LIN {X -102.468,Y -19.656,Z -60.794,A -90.000,B 90.000,C 0.000} C_DIS
LIN {X -102.647,Y -19.661,Z -60.638,A -90.000,B 90.000,C 0.000} C_DIS
LIN {X -103.007,Y -19.669,Z -60.305,A -90.000,B 90.000,C 0.000} C_DIS
LIN {X -103.209,Y -19.683,Z -60.113,A -90.000,B 90.000,C 0.000} C_DIS
LIN {X -103.495,Y -19.707,Z -59.844,A -90.000,B 90.000,C 0.000} C_DIS
LIN {X -103.666,Y -19.713,Z -59.667,A -90.000,B 90.000,C 0.000} C_DIS
LIN {X -103.779,Y -19.716,Z -59.547,A -90.000,B 90.000,C 0.000} C_DIS
LIN {X -103.860,Y -19.719,Z -59.459,A -90.000,B 90.000,C 0.000} C_DIS
LIN {X -104.495,Y -19.775,Z -58.745,A -90.000,B 90.000,C 0.000} C_DIS
LIN {X -104.595,Y -19.779,Z -58.623,A -90.000,B 90.000,C 0.000} C_DIS
LIN {X -104.835,Y -19.785,Z -58.316,A -90.000,B 90.000,C 0.000} C_DIS
LIN {X -104.978,Y -19.797,Z -58.132,A -90.000,B 90.000,C 0.000} C_DIS
LIN {X -105.043,Y -19.805,Z -58.047,A -90.000,B 90.000,C 0.000} C_DIS
LIN {X -105.125,Y -19.819,Z -57.934,A -90.000,B 90.000,C 0.000} C_DIS
LIN {X -105.385,Y -19.857,Z -57.556,A -90.000,B 90.000,C 0.000} C_DIS
LIN {X -105.527,Y -19.870,Z -57.329,A -90.000,B 90.000,C 0.000} C_DIS
LIN {X -105.764,Y -19.897,Z -56.936,A -90.000,B 90.000,C 0.000} C_DIS
LIN {X -105.854,Y -19.911,Z -56.776,A -90.000,B 90.000,C 0.000} C_DIS
LIN {X -105.917,Y -19.926,Z -56.657,A -90.000,B 90.000,C 0.000} C_DIS
LIN {X -105.996,Y -19.941,Z -56.500,A -90.000,B 90.000,C 0.000} C_DIS
LIN {X -106.032,Y -19.946,Z -56.422,A -90.000,B 90.000,C 0.000} C_DIS
LIN {X -106.214,Y -19.970,Z -56.038,A -90.000,B 90.000,C 0.000} C_DIS
LIN {X -106.380,Y -19.996,Z -55.650,A -90.000,B 90.000,C 0.000} C_DIS
LIN {X -106.472,Y -20.020,Z -55.411,A -90.000,B 90.000,C 0.000} C_DIS
LIN {X -106.494,Y -20.024,Z -55.349,A -90.000,B 90.000,C 0.000} C_DIS
LIN {X -106.535,Y -20.035,Z -55.220,A -90.000,B 90.000,C 0.000} C_DIS
LIN {X -106.617,Y -20.062,Z -54.946,A -90.000,B 90.000,C 0.000} C_DIS
LIN {X -106.692,Y -20.075,Z -54.624,A -90.000,B 90.000,C 0.000} C_DIS
LIN {X -106.760,Y -20.092,Z -54.341,A -90.000,B 90.000,C 0.000} C_DIS
LIN {X -106.862,Y -20.115,Z -53.878,A -90.000,B 90.000,C 0.000} C_DIS
LIN {X -106.884,Y -20.121,Z -53.754,A -90.000,B 90.000,C 0.000} C_DIS
LIN {X -106.893,Y -20.125,Z -53.683,A -90.000,B 90.000,C 0.000} C_DIS
LIN {X -106.930,Y -20.149,Z -53.353,A -90.000,B 90.000,C 0.000} C_DIS
LIN {X -106.945,Y -20.158,Z -53.148,A -90.000,B 90.000,C 0.000} C_DIS
LIN {X -106.963,Y -20.175,Z -52.914,A -90.000,B 90.000,C 0.000} C_DIS
LIN {X -106.986,Y -20.187,Z -52.670,A -90.000,B 90.000,C 0.000} C_DIS
LIN {X -106.991,Y -20.199,Z -52.434,A -90.000,B 90.000,C 0.000} C_DIS
LIN {X -106.989,Y -20.206,Z -52.353,A -90.000,B 90.000,C 0.000} C_DIS
LIN {X -106.977,Y -20.220,Z -52.109,A -90.000,B 90.000,C 0.000} C_DIS
LIN {X -106.972,Y -20.227,Z -51.945,A -90.000,B 90.000,C 0.000} C_DIS
LIN {X -106.965,Y -20.243,Z -51.722,A -90.000,B 90.000,C 0.000} C_DIS
LIN {X -106.951,Y -20.255,Z -51.466,A -90.000,B 90.000,C 0.000} C_DIS
LIN {X -106.935,Y -20.264,Z -51.321,A -90.000,B 90.000,C 0.000} C_DIS
LIN {X -106.911,Y -20.273,Z -51.181,A -90.000,B 90.000,C 0.000} C_DIS
LIN {X -106.852,Y -20.297,Z -50.866,A -90.000,B 90.000,C 0.000} C_DIS
LIN {X -106.771,Y -20.330,Z -50.476,A -90.000,B 90.000,C 0.000} C_DIS
LIN {X -106.685,Y -20.335,Z -50.140,A -90.000,B 90.000,C 0.000} C_DIS
LIN {X -106.782,Y -20.243,Z -49.888,A -90.000,B 90.000,C 0.000} C_DIS
LIN {X -106.856,Y -20.158,Z -49.671,A -90.000,B 90.000,C 0.000} C_DIS
LIN {X -106.932,Y -20.067,Z -49.428,A -90.000,B 90.000,C 0.000} C_DIS
LIN {X -106.948,Y -20.044,Z -49.370,A -90.000,B 90.000,C 0.000} C_DIS
LIN {X -106.980,Y -19.994,Z -49.227,A -90.000,B 90.000,C 0.000} C_DIS
LIN {X -107.015,Y -19.922,Z -49.018,A -90.000,B 90.000,C 0.000} C_DIS
LIN {X -107.031,Y -19.869,Z -48.872,A -90.000,B 90.000,C 0.000} C_DIS
LIN {X -107.043,Y -19.802,Z -48.689,A -90.000,B 90.000,C 0.000} C_DIS
LIN {X -107.043,Y -19.769,Z -48.600,A -90.000,B 90.000,C 0.000} C_DIS
LIN {X -107.040,Y -19.702,Z -48.416,A -90.000,B 90.000,C 0.000} C_DIS
LIN {X -107.158,Y -19.716,Z -48.219,A -90.000,B 90.000,C 0.000} C_DIS
LIN {X -107.387,Y -19.753,Z -47.792,A -90.000,B 90.000,C 0.000} C_DIS
LIN {X -107.530,Y -19.779,Z -47.517,A -90.000,B 90.000,C 0.000} C_DIS
LIN {X -107.589,Y -19.788,Z -47.393,A -90.000,B 90.000,C 0.000} C_DIS
LIN {X -107.781,Y -19.805,Z -46.947,A -90.000,B 90.000,C 0.000} C_DIS
LIN {X -107.936,Y -19.835,Z -46.542,A -90.000,B 90.000,C 0.000} C_DIS
LIN {X -108.076,Y -19.861,Z -46.147,A -90.000,B 90.000,C 0.000} C_DIS
LIN {X -108.110,Y -19.866,Z -46.039,A -90.000,B 90.000,C 0.000} C_DIS
LIN {X -108.258,Y -19.905,Z -45.517,A -90.000,B 90.000,C 0.000} C_DIS
LIN {X -108.292,Y -19.918,Z -45.382,A -90.000,B 90.000,C 0.000} C_DIS
LIN {X -108.367,Y -19.945,Z -44.989,A -90.000,B 90.000,C 0.000} C_DIS
LIN {X -108.401,Y -19.963,Z -44.786,A -90.000,B 90.000,C 0.000} C_DIS
LIN {X -108.450,Y -19.994,Z -44.452,A -90.000,B 90.000,C 0.000} C_DIS
LIN {X -108.458,Y -20.003,Z -44.374,A -90.000,B 90.000,C 0.000} C_DIS
LIN {X -108.475,Y -20.034,Z -44.027,A -90.000,B 90.000,C 0.000} C_DIS
LIN {X -108.482,Y -20.061,Z -43.676,A -90.000,B 90.000,C 0.000} C_DIS
LIN {X -108.481,Y -20.063,Z -43.623,A -90.000,B 90.000,C 0.000} C_DIS
LIN {X -108.472,Y -20.076,Z -43.437,A -90.000,B 90.000,C 0.000} C_DIS
LIN {X -108.460,Y -20.088,Z -43.312,A -90.000,B 90.000,C 0.000} C_DIS
LIN {X -108.430,Y -20.106,Z -43.070,A -90.000,B 90.000,C 0.000} C_DIS
LIN {X -108.391,Y -20.124,Z -42.770,A -90.000,B 90.000,C 0.000} C_DIS
LIN {X -108.369,Y -20.134,Z -42.620,A -90.000,B 90.000,C 0.000} C_DIS
LIN {X -108.351,Y -20.143,Z -42.521,A -90.000,B 90.000,C 0.000} C_DIS
LIN {X -108.295,Y -20.154,Z -42.273,A -90.000,B 90.000,C 0.000} C_DIS
LIN {X -108.254,Y -20.164,Z -42.113,A -90.000,B 90.000,C 0.000} C_DIS
LIN {X -108.187,Y -20.183,Z -41.874,A -90.000,B 90.000,C 0.000} C_DIS
LIN {X -108.175,Y -20.184,Z -41.836,A -90.000,B 90.000,C 0.000} C_DIS
LIN {X -108.036,Y -20.196,Z -41.450,A -90.000,B 90.000,C 0.000} C_DIS
LIN {X -107.992,Y -20.202,Z -41.337,A -90.000,B 90.000,C 0.000} C_DIS
LIN {X -107.941,Y -20.210,Z -41.219,A -90.000,B 90.000,C 0.000} C_DIS
LIN {X -107.830,Y -20.216,Z -40.993,A -90.000,B 90.000,C 0.000} C_DIS
LIN {X -107.652,Y -20.229,Z -40.655,A -90.000,B 90.000,C 0.000} C_DIS
LIN {X -107.557,Y -20.231,Z -40.499,A -90.000,B 90.000,C 0.000} C_DIS
LIN {X -107.486,Y -20.236,Z -40.390,A -90.000,B 90.000,C 0.000} C_DIS
LIN {X -107.378,Y -20.243,Z -40.218,A -90.000,B 90.000,C 0.000} C_DIS
LIN {X -107.336,Y -20.247,Z -40.156,A -90.000,B 90.000,C 0.000} C_DIS
LIN {X -107.134,Y -20.247,Z -39.892,A -90.000,B 90.000,C 0.000} C_DIS
LIN {X -106.995,Y -20.248,Z -39.727,A -90.000,B 90.000,C 0.000} C_DIS
LIN {X -106.913,Y -20.255,Z -39.638,A -90.000,B 90.000,C 0.000} C_DIS
LIN {X -106.815,Y -20.255,Z -39.541,A -90.000,B 90.000,C 0.000} C_DIS
LIN {X -106.736,Y -20.252,Z -39.457,A -90.000,B 90.000,C 0.000} C_DIS
LIN {X -106.666,Y -20.252,Z -39.388,A -90.000,B 90.000,C 0.000} C_DIS
LIN {X -106.465,Y -20.238,Z -39.204,A -90.000,B 90.000,C 0.000} C_DIS
LIN {X -106.419,Y -20.237,Z -39.161,A -90.000,B 90.000,C 0.000} C_DIS
LIN {X -106.281,Y -20.233,Z -39.052,A -90.000,B 90.000,C 0.000} C_DIS
LIN {X -106.141,Y -20.233,Z -38.949,A -90.000,B 90.000,C 0.000} C_DIS
LIN {X -106.028,Y -20.228,Z -38.869,A -90.000,B 90.000,C 0.000} C_DIS
LIN {X -105.932,Y -20.222,Z -38.807,A -90.000,B 90.000,C 0.000} C_DIS
LIN {X -105.709,Y -20.209,Z -38.671,A -90.000,B 90.000,C 0.000} C_DIS
LIN {X -105.617,Y -20.200,Z -38.618,A -90.000,B 90.000,C 0.000} C_DIS
LIN {X -105.493,Y -20.190,Z -38.549,A -90.000,B 90.000,C 0.000} C_DIS
LIN {X -105.295,Y -20.180,Z -38.450,A -90.000,B 90.000,C 0.000} C_DIS
LIN {X -105.169,Y -20.170,Z -38.390,A -90.000,B 90.000,C 0.000} C_DIS
LIN {X -104.969,Y -20.158,Z -38.302,A -90.000,B 90.000,C 0.000} C_DIS
LIN {X -104.908,Y -20.152,Z -38.281,A -90.000,B 90.000,C 0.000} C_DIS
LIN {X -104.636,Y -20.132,Z -38.197,A -90.000,B 90.000,C 0.000} C_DIS
LIN {X -104.324,Y -20.111,Z -38.104,A -90.000,B 90.000,C 0.000} C_DIS
LIN {X -104.248,Y -20.104,Z -38.084,A -90.000,B 90.000,C 0.000} C_DIS
LIN {X -104.041,Y -20.090,Z -38.032,A -90.000,B 90.000,C 0.000} C_DIS
LIN {X -103.918,Y -20.081,Z -38.000,A -90.000,B 90.000,C 0.000} C_DIS
LIN {X -103.778,Y -20.066,Z -37.966,A -90.000,B 90.000,C 0.000} C_DIS
LIN {X -103.743,Y -20.075,Z -37.948,A -90.000,B 90.000,C 0.000} C_DIS
LIN {X -103.593,Y -20.116,Z -37.876,A -90.000,B 90.000,C 0.000} C_DIS
LIN {X -103.525,Y -20.135,Z -37.847,A -90.000,B 90.000,C 0.000} C_DIS
LIN {X -103.189,Y -20.234,Z -37.708,A -90.000,B 90.000,C 0.000} C_DIS
LIN {X -103.098,Y -20.260,Z -37.678,A -90.000,B 90.000,C 0.000} C_DIS
LIN {X -102.820,Y -20.336,Z -37.593,A -90.000,B 90.000,C 0.000} C_DIS
LIN {X -102.445,Y -20.444,Z -37.498,A -90.000,B 90.000,C 0.000} C_DIS
LIN {X -102.298,Y -20.487,Z -37.465,A -90.000,B 90.000,C 0.000} C_DIS
LIN {X -102.220,Y -20.485,Z -37.368,A -90.000,B 90.000,C 0.000} C_DIS
LIN {X -102.027,Y -20.483,Z -37.139,A -90.000,B 90.000,C 0.000} C_DIS
LIN {X -101.812,Y -20.465,Z -36.903,A -90.000,B 90.000,C 0.000} C_DIS
LIN {X -101.694,Y -20.455,Z -36.777,A -90.000,B 90.000,C 0.000} C_DIS
LIN {X -101.599,Y -20.451,Z -36.687,A -90.000,B 90.000,C 0.000} C_DIS
LIN {X -101.321,Y -20.445,Z -36.439,A -90.000,B 90.000,C 0.000} C_DIS
LIN {X -101.201,Y -20.438,Z -36.339,A -90.000,B 90.000,C 0.000} C_DIS
LIN {X -100.770,Y -20.415,Z -35.994,A -90.000,B 90.000,C 0.000} C_DIS
LIN {X -100.652,Y -20.410,Z -35.905,A -90.000,B 90.000,C 0.000} C_DIS
LIN {X -100.499,Y -20.406,Z -35.797,A -90.000,B 90.000,C 0.000} C_DIS
LIN {X -100.151,Y -20.388,Z -35.556,A -90.000,B 90.000,C 0.000} C_DIS
LIN {X -99.916,Y -20.381,Z -35.405,A -90.000,B 90.000,C 0.000} C_DIS
LIN {X -99.744,Y -20.377,Z -35.300,A -90.000,B 90.000,C 0.000} C_DIS
LIN {X -99.281,Y -20.363,Z -35.024,A -90.000,B 90.000,C 0.000} C_DIS
LIN {X -98.910,Y -20.352,Z -34.805,A -90.000,B 90.000,C 0.000} C_DIS
LIN {X -98.295,Y -20.344,Z -34.463,A -90.000,B 90.000,C 0.000} C_DIS
LIN {X -97.990,Y -20.342,Z -34.302,A -90.000,B 90.000,C 0.000} C_DIS
LIN {X -97.805,Y -20.337,Z -34.195,A -90.000,B 90.000,C 0.000} C_DIS
LIN {X -97.584,Y -20.328,Z -34.071,A -90.000,B 90.000,C 0.000} C_DIS
LIN {X -97.137,Y -20.320,Z -33.838,A -90.000,B 90.000,C 0.000} C_DIS
LIN {X -96.832,Y -20.314,Z -33.683,A -90.000,B 90.000,C 0.000} C_DIS
LIN {X -96.610,Y -20.308,Z -33.567,A -90.000,B 90.000,C 0.000} C_DIS
LIN {X -96.600,Y -20.286,Z -33.521,A -90.000,B 90.000,C 0.000} C_DIS
LIN {X -96.618,Y -20.295,Z -33.331,A -90.000,B 90.000,C 0.000} C_DIS
LIN {X -96.627,Y -20.305,Z -33.207,A -90.000,B 90.000,C 0.000} C_DIS
LIN {X -96.630,Y -20.322,Z -33.062,A -90.000,B 90.000,C 0.000} C_DIS
LIN {X -96.627,Y -20.328,Z -32.959,A -90.000,B 90.000,C 0.000} C_DIS
LIN {X -96.631,Y -20.329,Z -32.851,A -90.000,B 90.000,C 0.000} C_DIS
LIN {X -96.632,Y -20.333,Z -32.719,A -90.000,B 90.000,C 0.000} C_DIS
LIN {X -96.627,Y -20.331,Z -32.618,A -90.000,B 90.000,C 0.000} C_DIS
LIN {X -96.607,Y -20.330,Z -32.367,A -90.000,B 90.000,C 0.000} C_DIS
LIN {X -96.588,Y -20.322,Z -32.206,A -90.000,B 90.000,C 0.000} C_DIS
LIN {X -96.575,Y -20.319,Z -32.113,A -90.000,B 90.000,C 0.000} C_DIS
LIN {X -96.549,Y -20.317,Z -31.978,A -90.000,B 90.000,C 0.000} C_DIS
LIN {X -96.525,Y -20.324,Z -31.864,A -90.000,B 90.000,C 0.000} C_DIS
LIN {X -96.472,Y -20.326,Z -31.649,A -90.000,B 90.000,C 0.000} C_DIS
LIN {X -96.439,Y -20.328,Z -31.525,A -90.000,B 90.000,C 0.000} C_DIS
LIN {X -96.403,Y -20.326,Z -31.420,A -90.000,B 90.000,C 0.000} C_DIS
LIN {X -96.330,Y -20.307,Z -31.149,A -90.000,B 90.000,C 0.000} C_DIS
LIN {X -96.289,Y -20.298,Z -31.020,A -90.000,B 90.000,C 0.000} C_DIS
LIN {X -96.223,Y -20.292,Z -30.847,A -90.000,B 90.000,C 0.000} C_DIS
LIN {X -96.154,Y -20.291,Z -30.672,A -90.000,B 90.000,C 0.000} C_DIS
LIN {X -96.118,Y -20.285,Z -30.589,A -90.000,B 90.000,C 0.000} C_DIS
LIN {X -96.058,Y -20.279,Z -30.460,A -90.000,B 90.000,C 0.000} C_DIS
LIN {X -96.010,Y -20.277,Z -30.369,A -90.000,B 90.000,C 0.000} C_DIS
LIN {X -95.824,Y -20.245,Z -29.966,A -90.000,B 90.000,C 0.000} C_DIS
LIN {X -95.770,Y -20.241,Z -29.860,A -90.000,B 90.000,C 0.000} C_DIS
LIN {X -95.637,Y -20.227,Z -29.641,A -90.000,B 90.000,C 0.000} C_DIS
LIN {X -95.523,Y -20.215,Z -29.457,A -90.000,B 90.000,C 0.000} C_DIS
LIN {X -95.471,Y -20.215,Z -29.381,A -90.000,B 90.000,C 0.000} C_DIS
LIN {X -95.353,Y -20.211,Z -29.196,A -90.000,B 90.000,C 0.000} C_DIS
LIN {X -95.243,Y -20.197,Z -29.034,A -90.000,B 90.000,C 0.000} C_DIS
LIN {X -95.164,Y -20.190,Z -28.926,A -90.000,B 90.000,C 0.000} C_DIS
LIN {X -94.971,Y -20.177,Z -28.684,A -90.000,B 90.000,C 0.000} C_DIS
LIN {X -94.863,Y -20.172,Z -28.548,A -90.000,B 90.000,C 0.000} C_DIS
LIN {X -94.731,Y -20.163,Z -28.412,A -90.000,B 90.000,C 0.000} C_DIS
LIN {X -94.601,Y -20.160,Z -28.288,A -90.000,B 90.000,C 0.000} C_DIS
LIN {X -94.475,Y -20.153,Z -28.171,A -90.000,B 90.000,C 0.000} C_DIS
LIN {X -94.314,Y -20.151,Z -28.021,A -90.000,B 90.000,C 0.000} C_DIS
LIN {X -94.055,Y -20.125,Z -27.801,A -90.000,B 90.000,C 0.000} C_DIS
LIN {X -93.954,Y -20.114,Z -27.720,A -90.000,B 90.000,C 0.000} C_DIS
LIN {X -93.785,Y -20.104,Z -27.590,A -90.000,B 90.000,C 0.000} C_DIS
LIN {X -93.556,Y -20.075,Z -27.428,A -90.000,B 90.000,C 0.000} C_DIS
LIN {X -93.439,Y -20.063,Z -27.351,A -90.000,B 90.000,C 0.000} C_DIS
LIN {X -93.127,Y -20.040,Z -27.158,A -90.000,B 90.000,C 0.000} C_DIS
LIN {X -93.022,Y -20.034,Z -27.096,A -90.000,B 90.000,C 0.000} C_DIS
LIN {X -92.971,Y -20.029,Z -27.070,A -90.000,B 90.000,C 0.000} C_DIS
LIN {X -92.805,Y -20.021,Z -26.987,A -90.000,B 90.000,C 0.000} C_DIS
LIN {X -92.331,Y -19.981,Z -26.769,A -90.000,B 90.000,C 0.000} C_DIS
LIN {X -91.928,Y -19.956,Z -26.589,A -90.000,B 90.000,C 0.000} C_DIS
LIN {X -91.695,Y -19.940,Z -26.497,A -90.000,B 90.000,C 0.000} C_DIS
LIN {X -91.552,Y -19.927,Z -26.445,A -90.000,B 90.000,C 0.000} C_DIS
LIN {X -91.434,Y -19.921,Z -26.407,A -90.000,B 90.000,C 0.000} C_DIS
LIN {X -91.264,Y -19.922,Z -26.345,A -90.000,B 90.000,C 0.000} C_DIS
LIN {X -91.192,Y -19.919,Z -26.315,A -90.000,B 90.000,C 0.000} C_DIS
LIN {X -91.034,Y -19.911,Z -26.253,A -90.000,B 90.000,C 0.000} C_DIS
LIN {X -90.902,Y -19.902,Z -26.204,A -90.000,B 90.000,C 0.000} C_DIS
LIN {X -90.698,Y -19.867,Z -26.116,A -90.000,B 90.000,C 0.000} C_DIS
LIN {X -90.661,Y -19.863,Z -26.098,A -90.000,B 90.000,C 0.000} C_DIS
LIN {X -90.314,Y -19.805,Z -25.911,A -90.000,B 90.000,C 0.000} C_DIS
LIN {X -90.185,Y -19.779,Z -25.852,A -90.000,B 90.000,C 0.000} C_DIS
LIN {X -90.105,Y -19.764,Z -25.809,A -90.000,B 90.000,C 0.000} C_DIS
LIN {X -89.802,Y -19.720,Z -25.651,A -90.000,B 90.000,C 0.000} C_DIS
LIN {X -89.689,Y -19.701,Z -25.598,A -90.000,B 90.000,C 0.000} C_DIS
LIN {X -89.546,Y -19.681,Z -25.525,A -90.000,B 90.000,C 0.000} C_DIS
LIN {X -89.281,Y -19.641,Z -25.389,A -90.000,B 90.000,C 0.000} C_DIS
LIN {X -89.187,Y -19.632,Z -25.335,A -90.000,B 90.000,C 0.000} C_DIS
LIN {X -88.817,Y -19.594,Z -25.143,A -90.000,B 90.000,C 0.000} C_DIS
LIN {X -88.591,Y -19.569,Z -25.028,A -90.000,B 90.000,C 0.000} C_DIS
LIN {X -88.410,Y -19.554,Z -24.924,A -90.000,B 90.000,C 0.000} C_DIS
LIN {X -88.172,Y -19.533,Z -24.792,A -90.000,B 90.000,C 0.000} C_DIS
LIN {X -88.036,Y -19.523,Z -24.707,A -90.000,B 90.000,C 0.000} C_DIS
LIN {X -87.575,Y -19.491,Z -24.432,A -90.000,B 90.000,C 0.000} C_DIS
LIN {X -87.416,Y -19.486,Z -24.324,A -90.000,B 90.000,C 0.000} C_DIS
LIN {X -87.164,Y -19.473,Z -24.150,A -90.000,B 90.000,C 0.000} C_DIS
LIN {X -86.793,Y -19.466,Z -23.855,A -90.000,B 90.000,C 0.000} C_DIS
LIN {X -86.730,Y -19.468,Z -23.795,A -90.000,B 90.000,C 0.000} C_DIS
LIN {X -86.537,Y -19.469,Z -23.611,A -90.000,B 90.000,C 0.000} C_DIS
LIN {X -86.318,Y -19.481,Z -23.370,A -90.000,B 90.000,C 0.000} C_DIS
LIN {X -86.206,Y -19.483,Z -23.245,A -90.000,B 90.000,C 0.000} C_DIS
LIN {X -85.931,Y -19.501,Z -22.900,A -90.000,B 90.000,C 0.000} C_DIS
LIN {X -85.450,Y -19.527,Z -22.280,A -90.000,B 90.000,C 0.000} C_DIS
LIN {X -84.861,Y -19.552,Z -21.540,A -90.000,B 90.000,C 0.000} C_DIS
LIN {X -84.646,Y -19.565,Z -21.273,A -90.000,B 90.000,C 0.000} C_DIS
LIN {X -84.419,Y -19.582,Z -20.981,A -90.000,B 90.000,C 0.000} C_DIS
LIN {X -84.355,Y -19.586,Z -20.904,A -90.000,B 90.000,C 0.000} C_DIS
LIN {X -84.280,Y -19.596,Z -20.802,A -90.000,B 90.000,C 0.000} C_DIS
LIN {X -84.210,Y -19.604,Z -20.710,A -90.000,B 90.000,C 0.000} C_DIS
LIN {X -84.113,Y -19.625,Z -20.561,A -90.000,B 90.000,C 0.000} C_DIS
LIN {X -83.875,Y -19.667,Z -20.229,A -90.000,B 90.000,C 0.000} C_DIS
LIN {X -83.761,Y -19.686,Z -20.089,A -90.000,B 90.000,C 0.000} C_DIS
LIN {X -83.565,Y -19.718,Z -19.855,A -90.000,B 90.000,C 0.000} C_DIS
LIN {X -83.405,Y -19.736,Z -19.685,A -90.000,B 90.000,C 0.000} C_DIS
LIN {X -83.151,Y -19.771,Z -19.426,A -90.000,B 90.000,C 0.000} C_DIS
LIN {X -83.000,Y -19.792,Z -19.277,A -90.000,B 90.000,C 0.000} C_DIS
LIN {X -82.917,Y -19.798,Z -19.205,A -90.000,B 90.000,C 0.000} C_DIS
LIN {X -82.679,Y -19.814,Z -18.999,A -90.000,B 90.000,C 0.000} C_DIS
LIN {X -82.618,Y -19.818,Z -18.951,A -90.000,B 90.000,C 0.000} C_DIS
LIN {X -82.353,Y -19.825,Z -18.759,A -90.000,B 90.000,C 0.000} C_DIS
LIN {X -82.249,Y -19.827,Z -18.688,A -90.000,B 90.000,C 0.000} C_DIS
LIN {X -82.022,Y -19.835,Z -18.556,A -90.000,B 90.000,C 0.000} C_DIS
LIN {X -81.744,Y -19.845,Z -18.402,A -90.000,B 90.000,C 0.000} C_DIS
LIN {X -81.591,Y -19.856,Z -18.324,A -90.000,B 90.000,C 0.000} C_DIS
LIN {X -81.356,Y -19.872,Z -18.218,A -90.000,B 90.000,C 0.000} C_DIS
LIN {X -80.963,Y -19.878,Z -18.067,A -90.000,B 90.000,C 0.000} C_DIS
LIN {X -80.823,Y -19.875,Z -18.019,A -90.000,B 90.000,C 0.000} C_DIS
LIN {X -80.687,Y -19.875,Z -17.978,A -90.000,B 90.000,C 0.000} C_DIS
LIN {X -80.483,Y -19.882,Z -17.921,A -90.000,B 90.000,C 0.000} C_DIS
LIN {X -80.143,Y -19.891,Z -17.838,A -90.000,B 90.000,C 0.000} C_DIS
LIN {X -80.074,Y -19.891,Z -17.824,A -90.000,B 90.000,C 0.000} C_DIS
LIN {X -79.971,Y -19.891,Z -17.810,A -90.000,B 90.000,C 0.000} C_DIS
LIN {X -79.718,Y -19.897,Z -17.779,A -90.000,B 90.000,C 0.000} C_DIS
LIN {X -79.322,Y -19.900,Z -17.738,A -90.000,B 90.000,C 0.000} C_DIS
LIN {X -79.150,Y -19.903,Z -17.721,A -90.000,B 90.000,C 0.000} C_DIS
LIN {X -79.012,Y -19.900,Z -17.715,A -90.000,B 90.000,C 0.000} C_DIS
LIN {X -78.774,Y -19.905,Z -17.713,A -90.000,B 90.000,C 0.000} C_DIS
LIN {X -78.599,Y -19.909,Z -17.717,A -90.000,B 90.000,C 0.000} C_DIS
LIN {X -78.403,Y -19.912,Z -17.728,A -90.000,B 90.000,C 0.000} C_DIS
LIN {X -78.089,Y -19.927,Z -17.753,A -90.000,B 90.000,C 0.000} C_DIS
LIN {X -77.678,Y -19.933,Z -17.797,A -90.000,B 90.000,C 0.000} C_DIS
LIN {X -77.525,Y -19.934,Z -17.822,A -90.000,B 90.000,C 0.000} C_DIS
LIN {X -77.266,Y -19.938,Z -17.869,A -90.000,B 90.000,C 0.000} C_DIS
LIN {X -76.923,Y -19.951,Z -17.940,A -90.000,B 90.000,C 0.000} C_DIS
LIN {X -76.818,Y -19.954,Z -17.966,A -90.000,B 90.000,C 0.000} C_DIS
LIN {X -76.561,Y -19.967,Z -18.034,A -90.000,B 90.000,C 0.000} C_DIS
LIN {X -76.281,Y -19.971,Z -18.121,A -90.000,B 90.000,C 0.000} C_DIS
LIN {X -75.975,Y -19.976,Z -18.219,A -90.000,B 90.000,C 0.000} C_DIS
LIN {X -75.734,Y -19.987,Z -18.303,A -90.000,B 90.000,C 0.000} C_DIS
LIN {X -75.635,Y -19.994,Z -18.339,A -90.000,B 90.000,C 0.000} C_DIS
LIN {X -75.465,Y -20.005,Z -18.409,A -90.000,B 90.000,C 0.000} C_DIS
LIN {X -74.762,Y -20.027,Z -18.725,A -90.000,B 90.000,C 0.000} C_DIS
LIN {X -74.605,Y -20.034,Z -18.800,A -90.000,B 90.000,C 0.000} C_DIS
LIN {X -74.394,Y -20.048,Z -18.911,A -90.000,B 90.000,C 0.000} C_DIS
LIN {X -74.268,Y -20.054,Z -18.979,A -90.000,B 90.000,C 0.000} C_DIS
LIN {X -73.804,Y -20.064,Z -19.251,A -90.000,B 90.000,C 0.000} C_DIS
LIN {X -73.492,Y -20.076,Z -19.444,A -90.000,B 90.000,C 0.000} C_DIS
LIN {X -72.936,Y -20.103,Z -19.799,A -90.000,B 90.000,C 0.000} C_DIS
LIN {X -72.712,Y -20.106,Z -19.949,A -90.000,B 90.000,C 0.000} C_DIS
LIN {X -72.234,Y -20.123,Z -20.285,A -90.000,B 90.000,C 0.000} C_DIS
LIN {X -71.884,Y -20.137,Z -20.537,A -90.000,B 90.000,C 0.000} C_DIS
LIN {X -71.462,Y -20.145,Z -20.864,A -90.000,B 90.000,C 0.000} C_DIS
LIN {X -71.236,Y -20.154,Z -21.049,A -90.000,B 90.000,C 0.000} C_DIS
LIN {X -70.880,Y -20.173,Z -21.348,A -90.000,B 90.000,C 0.000} C_DIS
LIN {X -70.783,Y -20.175,Z -21.433,A -90.000,B 90.000,C 0.000} C_DIS
LIN {X -70.418,Y -20.180,Z -21.756,A -90.000,B 90.000,C 0.000} C_DIS
LIN {X -70.128,Y -20.183,Z -22.043,A -90.000,B 90.000,C 0.000} C_DIS
LIN {X -69.442,Y -20.206,Z -22.752,A -90.000,B 90.000,C 0.000} C_DIS
LIN {X -69.187,Y -20.202,Z -23.032,A -90.000,B 90.000,C 0.000} C_DIS
LIN {X -69.083,Y -20.202,Z -23.159,A -90.000,B 90.000,C 0.000} C_DIS
LIN {X -68.869,Y -20.210,Z -23.438,A -90.000,B 90.000,C 0.000} C_DIS
LIN {X -68.637,Y -20.225,Z -23.754,A -90.000,B 90.000,C 0.000} C_DIS
LIN {X -68.583,Y -20.230,Z -23.831,A -90.000,B 90.000,C 0.000} C_DIS
LIN {X -68.309,Y -20.252,Z -24.250,A -90.000,B 90.000,C 0.000} C_DIS
LIN {X -68.204,Y -20.256,Z -24.417,A -90.000,B 90.000,C 0.000} C_DIS
LIN {X -68.032,Y -20.246,Z -24.710,A -90.000,B 90.000,C 0.000} C_DIS
LIN {X -67.865,Y -20.243,Z -25.017,A -90.000,B 90.000,C 0.000} C_DIS
LIN {X -67.828,Y -20.241,Z -25.087,A -90.000,B 90.000,C 0.000} C_DIS
LIN {X -67.749,Y -20.242,Z -25.253,A -90.000,B 90.000,C 0.000} C_DIS
LIN {X -67.626,Y -20.257,Z -25.556,A -90.000,B 90.000,C 0.000} C_DIS
LIN {X -67.456,Y -20.266,Z -26.002,A -90.000,B 90.000,C 0.000} C_DIS
LIN {X -67.395,Y -20.268,Z -26.166,A -90.000,B 90.000,C 0.000} C_DIS
LIN {X -67.219,Y -20.281,Z -26.690,A -90.000,B 90.000,C 0.000} C_DIS
LIN {X -67.180,Y -20.281,Z -26.813,A -90.000,B 90.000,C 0.000} C_DIS
LIN {X -67.098,Y -20.285,Z -27.099,A -90.000,B 90.000,C 0.000} C_DIS
LIN {X -67.045,Y -20.286,Z -27.302,A -90.000,B 90.000,C 0.000} C_DIS
LIN {X -66.996,Y -20.291,Z -27.515,A -90.000,B 90.000,C 0.000} C_DIS
LIN {X -66.968,Y -20.291,Z -27.645,A -90.000,B 90.000,C 0.000} C_DIS
LIN {X -66.922,Y -20.295,Z -27.887,A -90.000,B 90.000,C 0.000} C_DIS
LIN {X -66.829,Y -20.314,Z -28.354,A -90.000,B 90.000,C 0.000} C_DIS
LIN {X -66.764,Y -20.323,Z -28.692,A -90.000,B 90.000,C 0.000} C_DIS
LIN {X -66.683,Y -20.332,Z -29.124,A -90.000,B 90.000,C 0.000} C_DIS
LIN {X -66.657,Y -20.338,Z -29.304,A -90.000,B 90.000,C 0.000} C_DIS
LIN {X -66.626,Y -20.341,Z -29.467,A -90.000,B 90.000,C 0.000} C_DIS
LIN {X -66.435,Y -20.418,Z -30.349,A -90.000,B 90.000,C 0.000} C_DIS
LIN {X -66.338,Y -20.418,Z -30.590,A -90.000,B 90.000,C 0.000} C_DIS
LIN {X -66.194,Y -20.462,Z -30.893,A -90.000,B 90.000,C 0.000} C_DIS
LIN {X -66.076,Y -20.458,Z -31.015,A -90.000,B 90.000,C 0.000} C_DIS
LIN {X -65.600,Y -20.441,Z -31.509,A -90.000,B 90.000,C 0.000} C_DIS
LIN {X -65.490,Y -20.453,Z -31.618,A -90.000,B 90.000,C 0.000} C_DIS
LIN {X -64.665,Y -20.443,Z -32.167,A -90.000,B 90.000,C 0.000} C_DIS
LIN {X -64.188,Y -20.434,Z -32.479,A -90.000,B 90.000,C 0.000} C_DIS
LIN {X -63.993,Y -20.442,Z -32.599,A -90.000,B 90.000,C 0.000} C_DIS
LIN {X -62.272,Y -20.445,Z -33.500,A -90.000,B 90.000,C 0.000} C_DIS
LIN {X -61.786,Y -20.460,Z -33.747,A -90.000,B 90.000,C 0.000} C_DIS
LIN {X -61.215,Y -20.465,Z -34.007,A -90.000,B 90.000,C 0.000} C_DIS
LIN {X -60.289,Y -20.472,Z -34.425,A -90.000,B 90.000,C 0.000} C_DIS
LIN {X -59.386,Y -20.492,Z -34.825,A -90.000,B 90.000,C 0.000} C_DIS
LIN {X -58.037,Y -20.501,Z -35.386,A -90.000,B 90.000,C 0.000} C_DIS
LIN {X -57.168,Y -20.523,Z -35.739,A -90.000,B 90.000,C 0.000} C_DIS
LIN {X -57.094,Y -20.524,Z -35.767,A -90.000,B 90.000,C 0.000} C_DIS
LIN {X -55.415,Y -20.538,Z -36.392,A -90.000,B 90.000,C 0.000} C_DIS
LIN {X -54.701,Y -20.556,Z -36.652,A -90.000,B 90.000,C 0.000} C_DIS
LIN {X -54.626,Y -20.558,Z -36.679,A -90.000,B 90.000,C 0.000} C_DIS
LIN {X -53.682,Y -20.569,Z -36.987,A -90.000,B 90.000,C 0.000} C_DIS
LIN {X -52.765,Y -20.574,Z -37.274,A -90.000,B 90.000,C 0.000} C_DIS
LIN {X -52.105,Y -20.586,Z -37.477,A -90.000,B 90.000,C 0.000} C_DIS
LIN {X -51.908,Y -20.592,Z -37.536,A -90.000,B 90.000,C 0.000} C_DIS
LIN {X -50.899,Y -20.615,Z -37.808,A -90.000,B 90.000,C 0.000} C_DIS
LIN {X -50.089,Y -20.631,Z -38.019,A -90.000,B 90.000,C 0.000} C_DIS
LIN {X -49.669,Y -20.648,Z -38.124,A -90.000,B 90.000,C 0.000} C_DIS
LIN {X -49.038,Y -20.686,Z -38.279,A -90.000,B 90.000,C 0.000} C_DIS
LIN {X -48.880,Y -20.694,Z -38.311,A -90.000,B 90.000,C 0.000} C_DIS
LIN {X -47.890,Y -20.783,Z -38.492,A -90.000,B 90.000,C 0.000} C_DIS
LIN {X -47.180,Y -20.861,Z -38.621,A -90.000,B 90.000,C 0.000} C_DIS
LIN {X -46.693,Y -20.938,Z -38.708,A -90.000,B 90.000,C 0.000} C_DIS
LIN {X -46.558,Y -20.932,Z -38.567,A -90.000,B 90.000,C 0.000} C_DIS
LIN {X -46.503,Y -20.926,Z -38.512,A -90.000,B 90.000,C 0.000} C_DIS
LIN {X -46.406,Y -20.917,Z -38.419,A -90.000,B 90.000,C 0.000} C_DIS
LIN {X -46.283,Y -20.902,Z -38.318,A -90.000,B 90.000,C 0.000} C_DIS
LIN {X -46.130,Y -20.888,Z -38.206,A -90.000,B 90.000,C 0.000} C_DIS
LIN {X -45.841,Y -20.894,Z -37.988,A -90.000,B 90.000,C 0.000} C_DIS
LIN {X -45.672,Y -20.895,Z -37.866,A -90.000,B 90.000,C 0.000} C_DIS
LIN {X -45.583,Y -20.883,Z -37.771,A -90.000,B 90.000,C 0.000} C_DIS
LIN {X -45.528,Y -20.876,Z -37.717,A -90.000,B 90.000,C 0.000} C_DIS
LIN {X -45.447,Y -20.862,Z -37.647,A -90.000,B 90.000,C 0.000} C_DIS
LIN {X -45.399,Y -20.854,Z -37.609,A -90.000,B 90.000,C 0.000} C_DIS
LIN {X -45.179,Y -20.821,Z -37.452,A -90.000,B 90.000,C 0.000} C_DIS
LIN {X -45.044,Y -20.798,Z -37.362,A -90.000,B 90.000,C 0.000} C_DIS
LIN {X -45.002,Y -20.792,Z -37.337,A -90.000,B 90.000,C 0.000} C_DIS
LIN {X -44.923,Y -20.787,Z -37.292,A -90.000,B 90.000,C 0.000} C_DIS
LIN {X -44.811,Y -20.783,Z -37.235,A -90.000,B 90.000,C 0.000} C_DIS
LIN {X -44.570,Y -20.777,Z -37.126,A -90.000,B 90.000,C 0.000} C_DIS
LIN {X -44.300,Y -20.776,Z -37.025,A -90.000,B 90.000,C 0.000} C_DIS
LIN {X -43.832,Y -20.780,Z -36.907,A -90.000,B 90.000,C 0.000} C_DIS
LIN {X -43.705,Y -20.781,Z -36.876,A -90.000,B 90.000,C 0.000} C_DIS
LIN {X -43.612,Y -20.777,Z -36.854,A -90.000,B 90.000,C 0.000} C_DIS
LIN {X -43.394,Y -20.744,Z -36.738,A -90.000,B 90.000,C 0.000} C_DIS
LIN {X -43.300,Y -20.730,Z -36.691,A -90.000,B 90.000,C 0.000} C_DIS
LIN {X -43.030,Y -20.691,Z -36.579,A -90.000,B 90.000,C 0.000} C_DIS
LIN {X -42.805,Y -20.664,Z -36.499,A -90.000,B 90.000,C 0.000} C_DIS
LIN {X -42.674,Y -20.653,Z -36.465,A -90.000,B 90.000,C 0.000} C_DIS
LIN {X -42.114,Y -20.612,Z -36.328,A -90.000,B 90.000,C 0.000} C_DIS
LIN {X -41.835,Y -20.599,Z -36.279,A -90.000,B 90.000,C 0.000} C_DIS
LIN {X -41.552,Y -20.594,Z -36.249,A -90.000,B 90.000,C 0.000} C_DIS
LIN {X -40.756,Y -20.586,Z -36.178,A -90.000,B 90.000,C 0.000} C_DIS
LIN {X -40.532,Y -20.577,Z -36.160,A -90.000,B 90.000,C 0.000} C_DIS
LIN {X -39.872,Y -20.548,Z -36.101,A -90.000,B 90.000,C 0.000} C_DIS
LIN {X -38.785,Y -20.507,Z -36.002,A -90.000,B 90.000,C 0.000} C_DIS
LIN {X -38.643,Y -20.504,Z -35.993,A -90.000,B 90.000,C 0.000} C_DIS
LIN {X -37.788,Y -20.498,Z -35.971,A -90.000,B 90.000,C 0.000} C_DIS
LIN {X -37.534,Y -20.498,Z -35.967,A -90.000,B 90.000,C 0.000} C_DIS
LIN {X -36.686,Y -20.480,Z -35.964,A -90.000,B 90.000,C 0.000} C_DIS
LIN {X -36.086,Y -20.472,Z -35.970,A -90.000,B 90.000,C 0.000} C_DIS
LIN {X -33.666,Y -20.431,Z -36.001,A -90.000,B 90.000,C 0.000} C_DIS
LIN {X -33.504,Y -20.429,Z -36.006,A -90.000,B 90.000,C 0.000} C_DIS
LIN {X -32.902,Y -20.431,Z -36.040,A -90.000,B 90.000,C 0.000} C_DIS
LIN {X -31.689,Y -20.428,Z -36.144,A -90.000,B 90.000,C 0.000} C_DIS
LIN {X -30.416,Y -20.416,Z -36.256,A -90.000,B 90.000,C 0.000} C_DIS
LIN {X -29.912,Y -20.407,Z -36.294,A -90.000,B 90.000,C 0.000} C_DIS
LIN {X -28.471,Y -20.394,Z -36.392,A -90.000,B 90.000,C 0.000} C_DIS
LIN {X -28.164,Y -20.389,Z -36.414,A -90.000,B 90.000,C 0.000} C_DIS
LIN {X -27.915,Y -20.387,Z -36.435,A -90.000,B 90.000,C 0.000} C_DIS
LIN {X -27.784,Y -20.385,Z -36.443,A -90.000,B 90.000,C 0.000} C_DIS
LIN {X -27.409,Y -20.383,Z -36.475,A -90.000,B 90.000,C 0.000} C_DIS
LIN {X -26.259,Y -20.395,Z -36.585,A -90.000,B 90.000,C 0.000} C_DIS
LIN {X -25.639,Y -20.385,Z -36.653,A -90.000,B 90.000,C 0.000} C_DIS
LIN {X -25.364,Y -20.371,Z -36.669,A -90.000,B 90.000,C 0.000} C_DIS
LIN {X -24.461,Y -20.343,Z -36.712,A -90.000,B 90.000,C 0.000} C_DIS
LIN {X -23.566,Y -20.323,Z -36.778,A -90.000,B 90.000,C 0.000} C_DIS
LIN {X -23.169,Y -20.305,Z -36.793,A -90.000,B 90.000,C 0.000} C_DIS
LIN {X -22.470,Y -20.280,Z -36.817,A -90.000,B 90.000,C 0.000} C_DIS
LIN {X -22.137,Y -20.277,Z -36.842,A -90.000,B 90.000,C 0.000} C_DIS
LIN {X -21.228,Y -20.260,Z -36.915,A -90.000,B 90.000,C 0.000} C_DIS
LIN {X -20.885,Y -20.255,Z -36.945,A -90.000,B 90.000,C 0.000} C_DIS
LIN {X -20.789,Y -20.253,Z -36.955,A -90.000,B 90.000,C 0.000} C_DIS
LIN {X -20.623,Y -20.247,Z -36.974,A -90.000,B 90.000,C 0.000} C_DIS
LIN {X -18.363,Y -20.178,Z -37.270,A -90.000,B 90.000,C 0.000} C_DIS
LIN {X -16.717,Y -20.126,Z -37.514,A -90.000,B 90.000,C 0.000} C_DIS
LIN {X -15.863,Y -20.095,Z -37.646,A -90.000,B 90.000,C 0.000} C_DIS
LIN {X -15.433,Y -20.088,Z -37.722,A -90.000,B 90.000,C 0.000} C_DIS
LIN {X -15.242,Y -20.088,Z -37.761,A -90.000,B 90.000,C 0.000} C_DIS
LIN {X -13.482,Y -20.029,Z -38.165,A -90.000,B 90.000,C 0.000} C_DIS
LIN {X -12.775,Y -20.018,Z -38.334,A -90.000,B 90.000,C 0.000} C_DIS
LIN {X -12.207,Y -20.007,Z -38.468,A -90.000,B 90.000,C 0.000} C_DIS
LIN {X -12.014,Y -20.002,Z -38.515,A -90.000,B 90.000,C 0.000} C_DIS
LIN {X -11.342,Y -19.992,Z -38.696,A -90.000,B 90.000,C 0.000} C_DIS
LIN {X -10.679,Y -19.978,Z -38.877,A -90.000,B 90.000,C 0.000} C_DIS
LIN {X -9.593,Y -19.950,Z -39.170,A -90.000,B 90.000,C 0.000} C_DIS
LIN {X -8.895,Y -19.926,Z -39.363,A -90.000,B 90.000,C 0.000} C_DIS
LIN {X -8.780,Y -19.924,Z -39.396,A -90.000,B 90.000,C 0.000} C_DIS
LIN {X -7.783,Y -19.906,Z -39.717,A -90.000,B 90.000,C 0.000} C_DIS
LIN {X -5.874,Y -19.877,Z -40.328,A -90.000,B 90.000,C 0.000} C_DIS
LIN {X -5.386,Y -19.871,Z -40.489,A -90.000,B 90.000,C 0.000} C_DIS
LIN {X -4.127,Y -19.870,Z -40.945,A -90.000,B 90.000,C 0.000} C_DIS
LIN {X -2.607,Y -19.881,Z -41.479,A -90.000,B 90.000,C 0.000} C_DIS
LIN {X -2.515,Y -19.884,Z -41.509,A -90.000,B 90.000,C 0.000} C_DIS
LIN {X -2.356,Y -19.893,Z -41.564,A -90.000,B 90.000,C 0.000} C_DIS
LIN {X -2.073,Y -19.905,Z -41.668,A -90.000,B 90.000,C 0.000} C_DIS
LIN {X -0.991,Y -19.960,Z -42.077,A -90.000,B 90.000,C 0.000} C_DIS
LIN {X -0.854,Y -19.973,Z -42.122,A -90.000,B 90.000,C 0.000} C_DIS
LIN {X 0.170,Y -20.080,Z -42.466,A -90.000,B 90.000,C 0.000} C_DIS
LIN {X 0.322,Y -20.093,Z -42.520,A -90.000,B 90.000,C 0.000} C_DIS
LIN {X 0.338,Y -20.095,Z -42.526,A -90.000,B 90.000,C 0.000} C_DIS
LIN {X 1.002,Y -20.165,Z -42.782,A -90.000,B 90.000,C 0.000} C_DIS
LIN {X 1.406,Y -20.226,Z -42.927,A -90.000,B 90.000,C 0.000} C_DIS
LIN {X 2.053,Y -20.328,Z -43.166,A -90.000,B 90.000,C 0.000} C_DIS
LIN {X 2.520,Y -20.388,Z -43.349,A -90.000,B 90.000,C 0.000} C_DIS
LIN {X 2.816,Y -20.425,Z -43.461,A -90.000,B 90.000,C 0.000} C_DIS
LIN {X 3.142,Y -20.482,Z -43.573,A -90.000,B 90.000,C 0.000} C_DIS
LIN {X 3.189,Y -20.489,Z -43.588,A -90.000,B 90.000,C 0.000} C_DIS
LIN {X 3.380,Y -20.522,Z -43.651,A -90.000,B 90.000,C 0.000} C_DIS
LIN {X 3.890,Y -20.553,Z -43.692,A -90.000,B 90.000,C 0.000} C_DIS
LIN {X 4.350,Y -20.586,Z -43.744,A -90.000,B 90.000,C 0.000} C_DIS
LIN {X 4.688,Y -20.578,Z -43.705,A -90.000,B 90.000,C 0.000} C_DIS
LIN {X 5.057,Y -20.569,Z -43.621,A -90.000,B 90.000,C 0.000} C_DIS
LIN {X 5.587,Y -20.544,Z -43.506,A -90.000,B 90.000,C 0.000} C_DIS
LIN {X 5.963,Y -20.537,Z -43.445,A -90.000,B 90.000,C 0.000} C_DIS
LIN {X 7.136,Y -20.473,Z -43.173,A -90.000,B 90.000,C 0.000} C_DIS
LIN {X 7.495,Y -20.455,Z -43.096,A -90.000,B 90.000,C 0.000} C_DIS
LIN {X 7.927,Y -20.436,Z -43.009,A -90.000,B 90.000,C 0.000} C_DIS
LIN {X 8.066,Y -20.426,Z -42.974,A -90.000,B 90.000,C 0.000} C_DIS
LIN {X 8.462,Y -20.391,Z -42.879,A -90.000,B 90.000,C 0.000} C_DIS
LIN {X 8.548,Y -20.384,Z -42.860,A -90.000,B 90.000,C 0.000} C_DIS
LIN {X 8.856,Y -20.364,Z -42.800,A -90.000,B 90.000,C 0.000} C_DIS
LIN {X 9.329,Y -20.335,Z -42.714,A -90.000,B 90.000,C 0.000} C_DIS
LIN {X 9.627,Y -20.308,Z -42.667,A -90.000,B 90.000,C 0.000} C_DIS
LIN {X 10.629,Y -20.245,Z -42.533,A -90.000,B 90.000,C 0.000} C_DIS
LIN {X 11.090,Y -20.204,Z -42.476,A -90.000,B 90.000,C 0.000} C_DIS
LIN {X 11.189,Y -20.197,Z -42.466,A -90.000,B 90.000,C 0.000} C_DIS
LIN {X 12.075,Y -20.148,Z -42.395,A -90.000,B 90.000,C 0.000} C_DIS
LIN {X 12.960,Y -20.084,Z -42.338,A -90.000,B 90.000,C 0.000} C_DIS
LIN {X 13.059,Y -20.078,Z -42.334,A -90.000,B 90.000,C 0.000} C_DIS
LIN {X 13.305,Y -20.067,Z -42.323,A -90.000,B 90.000,C 0.000} C_DIS
LIN {X 14.277,Y -20.033,Z -42.285,A -90.000,B 90.000,C 0.000} C_DIS
LIN {X 15.117,Y -19.997,Z -42.259,A -90.000,B 90.000,C 0.000} C_DIS
LIN {X 15.806,Y -19.968,Z -42.241,A -90.000,B 90.000,C 0.000} C_DIS
LIN {X 16.322,Y -19.953,Z -42.234,A -90.000,B 90.000,C 0.000} C_DIS
LIN {X 17.039,Y -19.928,Z -42.221,A -90.000,B 90.000,C 0.000} C_DIS
LIN {X 17.245,Y -19.918,Z -42.220,A -90.000,B 90.000,C 0.000} C_DIS
LIN {X 18.467,Y -19.881,Z -42.193,A -90.000,B 90.000,C 0.000} C_DIS
LIN {X 19.527,Y -19.847,Z -42.173,A -90.000,B 90.000,C 0.000} C_DIS
LIN {X 19.735,Y -19.843,Z -42.166,A -90.000,B 90.000,C 0.000} C_DIS
LIN {X 20.611,Y -19.837,Z -42.137,A -90.000,B 90.000,C 0.000} C_DIS
LIN {X 21.646,Y -19.809,Z -42.085,A -90.000,B 90.000,C 0.000} C_DIS
LIN {X 22.225,Y -19.811,Z -42.042,A -90.000,B 90.000,C 0.000} C_DIS
LIN {X 22.981,Y -19.821,Z -41.977,A -90.000,B 90.000,C 0.000} C_DIS
LIN {X 23.822,Y -19.808,Z -41.883,A -90.000,B 90.000,C 0.000} C_DIS
LIN {X 24.730,Y -19.823,Z -41.747,A -90.000,B 90.000,C 0.000} C_DIS
LIN {X 24.891,Y -19.820,Z -41.717,A -90.000,B 90.000,C 0.000} C_DIS
LIN {X 25.407,Y -19.816,Z -41.617,A -90.000,B 90.000,C 0.000} C_DIS
LIN {X 25.783,Y -19.810,Z -41.546,A -90.000,B 90.000,C 0.000} C_DIS
LIN {X 26.742,Y -19.823,Z -41.324,A -90.000,B 90.000,C 0.000} C_DIS
LIN {X 26.810,Y -19.822,Z -41.306,A -90.000,B 90.000,C 0.000} C_DIS
LIN {X 27.704,Y -19.797,Z -41.085,A -90.000,B 90.000,C 0.000} C_DIS
LIN {X 28.417,Y -19.790,Z -40.893,A -90.000,B 90.000,C 0.000} C_DIS
LIN {X 28.733,Y -19.787,Z -40.809,A -90.000,B 90.000,C 0.000} C_DIS
LIN {X 29.420,Y -19.769,Z -40.614,A -90.000,B 90.000,C 0.000} C_DIS
LIN {X 30.020,Y -19.737,Z -40.464,A -90.000,B 90.000,C 0.000} C_DIS
LIN {X 30.151,Y -19.735,Z -40.426,A -90.000,B 90.000,C 0.000} C_DIS
LIN {X 30.855,Y -19.733,Z -40.228,A -90.000,B 90.000,C 0.000} C_DIS
LIN {X 31.123,Y -19.725,Z -40.163,A -90.000,B 90.000,C 0.000} C_DIS
LIN {X 31.611,Y -19.702,Z -40.037,A -90.000,B 90.000,C 0.000} C_DIS
LIN {X 32.156,Y -19.680,Z -39.902,A -90.000,B 90.000,C 0.000} C_DIS
LIN {X 32.582,Y -19.659,Z -39.807,A -90.000,B 90.000,C 0.000} C_DIS
LIN {X 33.485,Y -19.629,Z -39.596,A -90.000,B 90.000,C 0.000} C_DIS
LIN {X 34.112,Y -19.625,Z -39.460,A -90.000,B 90.000,C 0.000} C_DIS
LIN {X 34.317,Y -19.617,Z -39.427,A -90.000,B 90.000,C 0.000} C_DIS
LIN {X 34.766,Y -19.593,Z -39.352,A -90.000,B 90.000,C 0.000} C_DIS
LIN {X 35.154,Y -19.575,Z -39.289,A -90.000,B 90.000,C 0.000} C_DIS
LIN {X 35.518,Y -19.565,Z -39.220,A -90.000,B 90.000,C 0.000} C_DIS
LIN {X 36.078,Y -19.550,Z -39.139,A -90.000,B 90.000,C 0.000} C_DIS
LIN {X 36.635,Y -19.527,Z -39.075,A -90.000,B 90.000,C 0.000} C_DIS
LIN {X 37.054,Y -19.513,Z -39.029,A -90.000,B 90.000,C 0.000} C_DIS
LIN {X 37.486,Y -19.505,Z -38.988,A -90.000,B 90.000,C 0.000} C_DIS
LIN {X 38.015,Y -19.497,Z -38.944,A -90.000,B 90.000,C 0.000} C_DIS
LIN {X 38.549,Y -19.478,Z -38.930,A -90.000,B 90.000,C 0.000} C_DIS
LIN {X 39.054,Y -19.458,Z -38.924,A -90.000,B 90.000,C 0.000} C_DIS
LIN {X 39.644,Y -19.439,Z -38.917,A -90.000,B 90.000,C 0.000} C_DIS
LIN {X 40.081,Y -19.435,Z -38.916,A -90.000,B 90.000,C 0.000} C_DIS
LIN {X 40.520,Y -19.425,Z -38.935,A -90.000,B 90.000,C 0.000} C_DIS
LIN {X 41.151,Y -19.405,Z -38.982,A -90.000,B 90.000,C 0.000} C_DIS
LIN {X 41.751,Y -19.392,Z -39.029,A -90.000,B 90.000,C 0.000} C_DIS
LIN {X 42.149,Y -19.388,Z -39.062,A -90.000,B 90.000,C 0.000} C_DIS
LIN {X 42.660,Y -19.381,Z -39.124,A -90.000,B 90.000,C 0.000} C_DIS
LIN {X 43.083,Y -19.373,Z -39.196,A -90.000,B 90.000,C 0.000} C_DIS
LIN {X 43.733,Y -19.361,Z -39.314,A -90.000,B 90.000,C 0.000} C_DIS
LIN {X 44.368,Y -19.349,Z -39.447,A -90.000,B 90.000,C 0.000} C_DIS
LIN {X 44.792,Y -19.346,Z -39.536,A -90.000,B 90.000,C 0.000} C_DIS
LIN {X 45.274,Y -19.341,Z -39.651,A -90.000,B 90.000,C 0.000} C_DIS
LIN {X 45.605,Y -19.342,Z -39.731,A -90.000,B 90.000,C 0.000} C_DIS
LIN {X 46.072,Y -19.339,Z -39.868,A -90.000,B 90.000,C 0.000} C_DIS
LIN {X 46.451,Y -19.333,Z -40.000,A -90.000,B 90.000,C 0.000} C_DIS
LIN {X 47.384,Y -19.326,Z -40.325,A -90.000,B 90.000,C 0.000} C_DIS
LIN {X 48.446,Y -19.318,Z -40.738,A -90.000,B 90.000,C 0.000} C_DIS
LIN {X 48.983,Y -19.317,Z -40.947,A -90.000,B 90.000,C 0.000} C_DIS
LIN {X 49.433,Y -19.317,Z -41.131,A -90.000,B 90.000,C 0.000} C_DIS
LIN {X 49.690,Y -19.316,Z -41.256,A -90.000,B 90.000,C 0.000} C_DIS
LIN {X 50.922,Y -19.313,Z -41.874,A -90.000,B 90.000,C 0.000} C_DIS
LIN {X 52.074,Y -19.311,Z -42.483,A -90.000,B 90.000,C 0.000} C_DIS
LIN {X 52.542,Y -19.312,Z -42.736,A -90.000,B 90.000,C 0.000} C_DIS
LIN {X 53.767,Y -19.310,Z -43.515,A -90.000,B 90.000,C 0.000} C_DIS
LIN {X 55.062,Y -19.309,Z -44.321,A -90.000,B 90.000,C 0.000} C_DIS
LIN {X 55.465,Y -19.309,Z -44.596,A -90.000,B 90.000,C 0.000} C_DIS
LIN {X 55.827,Y -19.309,Z -44.867,A -90.000,B 90.000,C 0.000} C_DIS
LIN {X 56.621,Y -19.309,Z -45.440,A -90.000,B 90.000,C 0.000} C_DIS
LIN {X 57.716,Y -19.310,Z -46.253,A -90.000,B 90.000,C 0.000} C_DIS
LIN {X 58.900,Y -19.310,Z -47.253,A -90.000,B 90.000,C 0.000} C_DIS
LIN {X 60.073,Y -19.310,Z -48.267,A -90.000,B 90.000,C 0.000} C_DIS
LIN {X 61.789,Y -19.312,Z -49.790,A -90.000,B 90.000,C 0.000} C_DIS
LIN {X 62.556,Y -19.315,Z -50.412,A -90.000,B 90.000,C 0.000} C_DIS
LIN {X 62.753,Y -19.316,Z -50.576,A -90.000,B 90.000,C 0.000} C_DIS
LIN {X 63.481,Y -19.319,Z -51.192,A -90.000,B 90.000,C 0.000} C_DIS
LIN {X 63.730,Y -19.323,Z -51.374,A -90.000,B 90.000,C 0.000} C_DIS
LIN {X 64.732,Y -19.327,Z -52.104,A -90.000,B 90.000,C 0.000} C_DIS
LIN {X 65.188,Y -19.331,Z -52.430,A -90.000,B 90.000,C 0.000} C_DIS
LIN {X 65.379,Y -19.336,Z -52.549,A -90.000,B 90.000,C 0.000} C_DIS
LIN {X 65.992,Y -19.338,Z -52.930,A -90.000,B 90.000,C 0.000} C_DIS
LIN {X 66.614,Y -19.344,Z -53.298,A -90.000,B 90.000,C 0.000} C_DIS
LIN {X 67.735,Y -19.347,Z -53.955,A -90.000,B 90.000,C 0.000} C_DIS
LIN {X 69.379,Y -19.352,Z -54.893,A -90.000,B 90.000,C 0.000} C_DIS
LIN {X 71.571,Y -19.355,Z -56.195,A -90.000,B 90.000,C 0.000} C_DIS
LIN {X 73.574,Y -19.358,Z -57.514,A -90.000,B 90.000,C 0.000} C_DIS
LIN {X 73.975,Y -19.359,Z -57.782,A -90.000,B 90.000,C 0.000} C_DIS
LIN {X 75.171,Y -19.363,Z -58.730,A -90.000,B 90.000,C 0.000} C_DIS
LIN {X 75.696,Y -19.367,Z -59.141,A -90.000,B 90.000,C 0.000} C_DIS
LIN {X 75.964,Y -19.367,Z -59.362,A -90.000,B 90.000,C 0.000} C_DIS
LIN {X 76.068,Y -19.369,Z -59.449,A -90.000,B 90.000,C 0.000} C_DIS
LIN {X 77.012,Y -19.375,Z -60.331,A -90.000,B 90.000,C 0.000} C_DIS
LIN {X 77.512,Y -19.381,Z -60.786,A -90.000,B 90.000,C 0.000} C_DIS
LIN {X 77.833,Y -19.381,Z -61.105,A -90.000,B 90.000,C 0.000} C_DIS
LIN {X 78.164,Y -19.384,Z -61.461,A -90.000,B 90.000,C 0.000} C_DIS
LIN {X 78.925,Y -19.396,Z -62.254,A -90.000,B 90.000,C 0.000} C_DIS
LIN {X 78.991,Y -19.365,Z -62.309,A -90.000,B 90.000,C 0.000} C_DIS
LIN {X 79.130,Y -19.331,Z -62.438,A -90.000,B 90.000,C 0.000} C_DIS
LIN {X 79.194,Y -19.320,Z -62.510,A -90.000,B 90.000,C 0.000} C_DIS
LIN {X 79.323,Y -19.309,Z -62.659,A -90.000,B 90.000,C 0.000} C_DIS
LIN {X 79.360,Y -19.308,Z -62.702,A -90.000,B 90.000,C 0.000} C_DIS
LIN {X 79.360,Y -60.000,Z -62.702,A -90.000,B 90.000,C 0.000} C_DIS
LIN {X 92.113,Y -60.000,Z -43.585,A -90.000,B 90.000,C 0.000} C_DIS
LIN {X 92.113,Y -19.308,Z -43.585,A -90.000,B 90.000,C 0.000} C_DIS
LIN {X 92.210,Y -19.308,Z -43.517,A -90.000,B 90.000,C 0.000} C_DIS
LIN {X 92.210,Y -60.000,Z -43.517,A -90.000,B 90.000,C 0.000} C_DIS
LIN {X 111.588,Y -60.000,Z -35.186,A -90.000,B 90.000,C 0.000} C_DIS
LIN {X 111.588,Y -19.308,Z -35.186,A -90.000,B 90.000,C 0.000} C_DIS
LIN {X 111.754,Y -19.308,Z -35.218,A -90.000,B 90.000,C 0.000} C_DIS
LIN {X 111.754,Y -60.000,Z -35.218,A -90.000,B 90.000,C 0.000} C_DIS
LIN {X 117.203,Y -60.000,Z -45.931,A -90.000,B 90.000,C 0.000} C_DIS
LIN {X 117.203,Y -19.308,Z -45.931,A -90.000,B 90.000,C 0.000} C_DIS
LIN {X 117.196,Y -19.308,Z -45.955,A -90.000,B 90.000,C 0.000} C_DIS
LIN {X 117.196,Y -60.000,Z -45.955,A -90.000,B 90.000,C 0.000} C_DIS
LIN {X 111.259,Y -60.000,Z -60.448,A -90.000,B 90.000,C 0.000} C_DIS
LIN {X 111.259,Y -19.308,Z -60.448,A -90.000,B 90.000,C 0.000} C_DIS
LIN {X 111.207,Y -19.308,Z -60.638,A -90.000,B 90.000,C 0.000} C_DIS
LIN {X 111.207,Y -60.000,Z -60.638,A -90.000,B 90.000,C 0.000} C_DIS
LIN {X 99.852,Y -60.000,Z -87.230,A -90.000,B 90.000,C 0.000} C_DIS
LIN {X 99.852,Y -19.308,Z -87.230,A -90.000,B 90.000,C 0.000} C_DIS
LIN {X 99.858,Y -19.308,Z -87.310,A -90.000,B 90.000,C 0.000} C_DIS
LIN {X 99.887,Y -19.306,Z -87.679,A -90.000,B 90.000,C 0.000} C_DIS
LIN {X 99.891,Y -19.302,Z -87.732,A -90.000,B 90.000,C 0.000} C_DIS
LIN {X 99.896,Y -19.299,Z -87.739,A -90.000,B 90.000,C 0.000} C_DIS
LIN {X 99.918,Y -19.308,Z -88.154,A -90.000,B 90.000,C 0.000} C_DIS
LIN {X 99.971,Y -19.324,Z -88.905,A -90.000,B 90.000,C 0.000} C_DIS
LIN {X 99.996,Y -19.308,Z -89.262,A -90.000,B 90.000,C 0.000} C_DIS
LIN {X 99.996,Y -60.000,Z -89.262,A -90.000,B 90.000,C 0.000} C_DIS
LIN {X 1.187,Y -60.000,Z -40.890,A -90.000,B 90.000,C 0.000} C_DIS
LIN {X 1.187,Y -19.308,Z -40.890,A -90.000,B 90.000,C 0.000} C_DIS
LIN {X 2.149,Y -19.466,Z -41.234,A -90.000,B 90.000,C 0.000} C_DIS
LIN {X 2.936,Y -19.597,Z -41.522,A -90.000,B 90.000,C 0.000} C_DIS
LIN {X 3.324,Y -19.664,Z -41.665,A -90.000,B 90.000,C 0.000} C_DIS
LIN {X 3.824,Y -19.755,Z -41.839,A -90.000,B 90.000,C 0.000} C_DIS
LIN {X 3.831,Y -19.756,Z -41.841,A -90.000,B 90.000,C 0.000} C_DIS
LIN {X 4.149,Y -19.771,Z -41.870,A -90.000,B 90.000,C 0.000} C_DIS
LIN {X 4.365,Y -19.785,Z -41.895,A -90.000,B 90.000,C 0.000} C_DIS
LIN {X 5.164,Y -19.708,Z -41.740,A -90.000,B 90.000,C 0.000} C_DIS
LIN {X 5.277,Y -19.698,Z -41.721,A -90.000,B 90.000,C 0.000} C_DIS
LIN {X 5.588,Y -19.675,Z -41.678,A -90.000,B 90.000,C 0.000} C_DIS
LIN {X 6.725,Y -19.549,Z -41.448,A -90.000,B 90.000,C 0.000} C_DIS
LIN {X 7.106,Y -19.509,Z -41.377,A -90.000,B 90.000,C 0.000} C_DIS
LIN {X 7.487,Y -19.471,Z -41.312,A -90.000,B 90.000,C 0.000} C_DIS
LIN {X 7.681,Y -19.446,Z -41.270,A -90.000,B 90.000,C 0.000} C_DIS
LIN {X 7.874,Y -19.423,Z -41.227,A -90.000,B 90.000,C 0.000} C_DIS
LIN {X 8.106,Y -19.393,Z -41.180,A -90.000,B 90.000,C 0.000} C_DIS
LIN {X 8.305,Y -19.370,Z -41.147,A -90.000,B 90.000,C 0.000} C_DIS
LIN {X 8.550,Y -19.335,Z -41.111,A -90.000,B 90.000,C 0.000} C_DIS
LIN {X 8.751,Y -19.308,Z -41.084,A -90.000,B 90.000,C 0.000} C_DIS
LIN {X 8.751,Y -60.000,Z -41.084,A -90.000,B 90.000,C 0.000} C_DIS
LIN {X -65.145,Y -60.000,Z -27.947,A -90.000,B 90.000,C 0.000} C_DIS
LIN {X -65.145,Y -19.308,Z -27.947,A -90.000,B 90.000,C 0.000} C_DIS
LIN {X -65.078,Y -19.337,Z -28.231,A -90.000,B 90.000,C 0.000} C_DIS
LIN {X -64.944,Y -19.392,Z -28.819,A -90.000,B 90.000,C 0.000} C_DIS
LIN {X -64.896,Y -19.418,Z -29.064,A -90.000,B 90.000,C 0.000} C_DIS
LIN {X -64.680,Y -19.578,Z -29.848,A -90.000,B 90.000,C 0.000} C_DIS
LIN {X -64.662,Y -19.583,Z -29.887,A -90.000,B 90.000,C 0.000} C_DIS
LIN {X -64.497,Y -19.575,Z -30.059,A -90.000,B 90.000,C 0.000} C_DIS
LIN {X -64.320,Y -19.592,Z -30.227,A -90.000,B 90.000,C 0.000} C_DIS
LIN {X -63.681,Y -19.583,Z -30.653,A -90.000,B 90.000,C 0.000} C_DIS
LIN {X -63.412,Y -19.578,Z -30.829,A -90.000,B 90.000,C 0.000} C_DIS
LIN {X -63.082,Y -19.594,Z -31.031,A -90.000,B 90.000,C 0.000} C_DIS
LIN {X -62.599,Y -19.599,Z -31.282,A -90.000,B 90.000,C 0.000} C_DIS
LIN {X -61.852,Y -19.613,Z -31.666,A -90.000,B 90.000,C 0.000} C_DIS
LIN {X -60.978,Y -19.650,Z -32.105,A -90.000,B 90.000,C 0.000} C_DIS
LIN {X -60.311,Y -19.672,Z -32.402,A -90.000,B 90.000,C 0.000} C_DIS
LIN {X -60.031,Y -19.681,Z -32.525,A -90.000,B 90.000,C 0.000} C_DIS
LIN {X -58.646,Y -19.738,Z -33.127,A -90.000,B 90.000,C 0.000} C_DIS
LIN {X -58.368,Y -19.746,Z -33.240,A -90.000,B 90.000,C 0.000} C_DIS
LIN {X -57.866,Y -19.755,Z -33.446,A -90.000,B 90.000,C 0.000} C_DIS
LIN {X -56.480,Y -19.809,Z -34.002,A -90.000,B 90.000,C 0.000} C_DIS
LIN {X -55.538,Y -19.834,Z -34.346,A -90.000,B 90.000,C 0.000} C_DIS
LIN {X -55.381,Y -19.837,Z -34.404,A -90.000,B 90.000,C 0.000} C_DIS
LIN {X -54.004,Y -19.898,Z -34.896,A -90.000,B 90.000,C 0.000} C_DIS
LIN {X -53.100,Y -19.928,Z -35.184,A -90.000,B 90.000,C 0.000} C_DIS
LIN {X -52.946,Y -19.933,Z -35.231,A -90.000,B 90.000,C 0.000} C_DIS
LIN {X -52.133,Y -19.982,Z -35.470,A -90.000,B 90.000,C 0.000} C_DIS
LIN {X -51.366,Y -20.038,Z -35.692,A -90.000,B 90.000,C 0.000} C_DIS
LIN {X -50.343,Y -20.107,Z -35.954,A -90.000,B 90.000,C 0.000} C_DIS
LIN {X -50.119,Y -20.125,Z -36.009,A -90.000,B 90.000,C 0.000} C_DIS
LIN {X -49.866,Y -20.158,Z -36.068,A -90.000,B 90.000,C 0.000} C_DIS
LIN {X -49.421,Y -20.207,Z -36.173,A -90.000,B 90.000,C 0.000} C_DIS
LIN {X -48.580,Y -20.281,Z -36.374,A -90.000,B 90.000,C 0.000} C_DIS
LIN {X -48.480,Y -20.292,Z -36.393,A -90.000,B 90.000,C 0.000} C_DIS
LIN {X -47.455,Y -20.426,Z -36.572,A -90.000,B 90.000,C 0.000} C_DIS
LIN {X -47.253,Y -20.455,Z -36.608,A -90.000,B 90.000,C 0.000} C_DIS
LIN {X -47.219,Y -20.452,Z -36.583,A -90.000,B 90.000,C 0.000} C_DIS
LIN {X -46.969,Y -20.417,Z -36.407,A -90.000,B 90.000,C 0.000} C_DIS
LIN {X -46.865,Y -20.394,Z -36.310,A -90.000,B 90.000,C 0.000} C_DIS
LIN {X -46.700,Y -20.356,Z -36.173,A -90.000,B 90.000,C 0.000} C_DIS
LIN {X -46.581,Y -20.330,Z -36.083,A -90.000,B 90.000,C 0.000} C_DIS
LIN {X -46.495,Y -20.312,Z -36.023,A -90.000,B 90.000,C 0.000} C_DIS
LIN {X -46.297,Y -20.273,Z -35.886,A -90.000,B 90.000,C 0.000} C_DIS
LIN {X -46.165,Y -20.260,Z -35.796,A -90.000,B 90.000,C 0.000} C_DIS
LIN {X -46.047,Y -20.248,Z -35.721,A -90.000,B 90.000,C 0.000} C_DIS
LIN {X -45.871,Y -20.234,Z -35.620,A -90.000,B 90.000,C 0.000} C_DIS
LIN {X -45.805,Y -20.230,Z -35.585,A -90.000,B 90.000,C 0.000} C_DIS
LIN {X -45.613,Y -20.205,Z -35.496,A -90.000,B 90.000,C 0.000} C_DIS
LIN {X -45.371,Y -20.167,Z -35.398,A -90.000,B 90.000,C 0.000} C_DIS
LIN {X -45.234,Y -20.147,Z -35.347,A -90.000,B 90.000,C 0.000} C_DIS
LIN {X -44.960,Y -20.112,Z -35.257,A -90.000,B 90.000,C 0.000} C_DIS
LIN {X -44.838,Y -20.098,Z -35.222,A -90.000,B 90.000,C 0.000} C_DIS
LIN {X -44.703,Y -20.087,Z -35.190,A -90.000,B 90.000,C 0.000} C_DIS
LIN {X -44.329,Y -20.056,Z -35.109,A -90.000,B 90.000,C 0.000} C_DIS
LIN {X -44.136,Y -20.020,Z -35.019,A -90.000,B 90.000,C 0.000} C_DIS
LIN {X -43.832,Y -19.971,Z -34.894,A -90.000,B 90.000,C 0.000} C_DIS
LIN {X -43.730,Y -19.956,Z -34.855,A -90.000,B 90.000,C 0.000} C_DIS
LIN {X -43.505,Y -19.925,Z -34.777,A -90.000,B 90.000,C 0.000} C_DIS
LIN {X -43.358,Y -19.907,Z -34.732,A -90.000,B 90.000,C 0.000} C_DIS
LIN {X -43.071,Y -19.870,Z -34.665,A -90.000,B 90.000,C 0.000} C_DIS
LIN {X -42.606,Y -19.813,Z -34.561,A -90.000,B 90.000,C 0.000} C_DIS
LIN {X -42.464,Y -19.798,Z -34.534,A -90.000,B 90.000,C 0.000} C_DIS
LIN {X -42.138,Y -19.770,Z -34.484,A -90.000,B 90.000,C 0.000} C_DIS
LIN {X -41.978,Y -19.760,Z -34.468,A -90.000,B 90.000,C 0.000} C_DIS
LIN {X -41.661,Y -19.744,Z -34.440,A -90.000,B 90.000,C 0.000} C_DIS
LIN {X -40.703,Y -19.702,Z -34.370,A -90.000,B 90.000,C 0.000} C_DIS
LIN {X -40.017,Y -19.662,Z -34.313,A -90.000,B 90.000,C 0.000} C_DIS
LIN {X -39.414,Y -19.621,Z -34.268,A -90.000,B 90.000,C 0.000} C_DIS
LIN {X -38.909,Y -19.589,Z -34.229,A -90.000,B 90.000,C 0.000} C_DIS
LIN {X -38.696,Y -19.580,Z -34.220,A -90.000,B 90.000,C 0.000} C_DIS
LIN {X -37.813,Y -19.556,Z -34.207,A -90.000,B 90.000,C 0.000} C_DIS
LIN {X -37.561,Y -19.551,Z -34.206,A -90.000,B 90.000,C 0.000} C_DIS
LIN {X -36.681,Y -19.532,Z -34.203,A -90.000,B 90.000,C 0.000} C_DIS
LIN {X -36.485,Y -19.530,Z -34.205,A -90.000,B 90.000,C 0.000} C_DIS
LIN {X -34.453,Y -19.459,Z -34.251,A -90.000,B 90.000,C 0.000} C_DIS
LIN {X -33.632,Y -19.429,Z -34.271,A -90.000,B 90.000,C 0.000} C_DIS
LIN {X -33.402,Y -19.423,Z -34.280,A -90.000,B 90.000,C 0.000} C_DIS
LIN {X -32.758,Y -19.417,Z -34.322,A -90.000,B 90.000,C 0.000} C_DIS
LIN {X -31.897,Y -19.416,Z -34.395,A -90.000,B 90.000,C 0.000} C_DIS
LIN {X -30.566,Y -19.391,Z -34.521,A -90.000,B 90.000,C 0.000} C_DIS
LIN {X -30.292,Y -19.383,Z -34.548,A -90.000,B 90.000,C 0.000} C_DIS
LIN {X -29.703,Y -19.359,Z -34.600,A -90.000,B 90.000,C 0.000} C_DIS
LIN {X -28.643,Y -19.324,Z -34.689,A -90.000,B 90.000,C 0.000} C_DIS
LIN {X -28.253,Y -19.308,Z -34.723,A -90.000,B 90.000,C 0.000} C_DIS
LIN {X -28.253,Y -60.000,Z -34.723,A -90.000,B 90.000,C 0.000} C_DIS
LIN {X -52.998,Y -60.000,Z -33.215,A -90.000,B 90.000,C 0.000} C_DIS
LIN {X -52.998,Y -19.308,Z -33.215,A -90.000,B 90.000,C 0.000} C_DIS
LIN {X -52.861,Y -19.317,Z -33.258,A -90.000,B 90.000,C 0.000} C_DIS
LIN {X -52.504,Y -19.351,Z -33.364,A -90.000,B 90.000,C 0.000} C_DIS
LIN {X -50.824,Y -19.500,Z -33.844,A -90.000,B 90.000,C 0.000} C_DIS
LIN {X -50.195,Y -19.546,Z -34.004,A -90.000,B 90.000,C 0.000} C_DIS
LIN {X -50.064,Y -19.561,Z -34.035,A -90.000,B 90.000,C 0.000} C_DIS
LIN {X -48.915,Y -19.653,Z -34.319,A -90.000,B 90.000,C 0.000} C_DIS
LIN {X -48.616,Y -19.676,Z -34.391,A -90.000,B 90.000,C 0.000} C_DIS
LIN {X -48.126,Y -19.739,Z -34.503,A -90.000,B 90.000,C 0.000} C_DIS
LIN {X -47.765,Y -19.779,Z -34.568,A -90.000,B 90.000,C 0.000} C_DIS
LIN {X -47.625,Y -19.754,Z -34.470,A -90.000,B 90.000,C 0.000} C_DIS
LIN {X -47.469,Y -19.722,Z -34.363,A -90.000,B 90.000,C 0.000} C_DIS
LIN {X -47.288,Y -19.675,Z -34.248,A -90.000,B 90.000,C 0.000} C_DIS
LIN {X -47.071,Y -19.623,Z -34.121,A -90.000,B 90.000,C 0.000} C_DIS
LIN {X -46.862,Y -19.567,Z -34.016,A -90.000,B 90.000,C 0.000} C_DIS
LIN {X -46.668,Y -19.524,Z -33.925,A -90.000,B 90.000,C 0.000} C_DIS
LIN {X -46.416,Y -19.473,Z -33.818,A -90.000,B 90.000,C 0.000} C_DIS
LIN {X -46.104,Y -19.414,Z -33.695,A -90.000,B 90.000,C 0.000} C_DIS
LIN {X -45.952,Y -19.388,Z -33.642,A -90.000,B 90.000,C 0.000} C_DIS
LIN {X -45.558,Y -19.329,Z -33.517,A -90.000,B 90.000,C 0.000} C_DIS
LIN {X -45.431,Y -19.308,Z -33.482,A -90.000,B 90.000,C 0.000} C_DIS
LIN {X -45.431,Y -60.000,Z -33.482,A -90.000,B 90.000,C 0.000} C_DIS
LIN {X -104.250,Y -60.000,Z -36.167,A -90.000,B 90.000,C 0.000} C_DIS
LIN {X -104.250,Y -19.308,Z -36.167,A -90.000,B 90.000,C 0.000} C_DIS
LIN {X -104.095,Y -19.347,Z -36.099,A -90.000,B 90.000,C 0.000} C_DIS
LIN {X -103.946,Y -19.385,Z -36.039,A -90.000,B 90.000,C 0.000} C_DIS
LIN {X -103.687,Y -19.439,Z -35.941,A -90.000,B 90.000,C 0.000} C_DIS
LIN {X -103.613,Y -19.455,Z -35.915,A -90.000,B 90.000,C 0.000} C_DIS
LIN {X -103.427,Y -19.498,Z -35.858,A -90.000,B 90.000,C 0.000} C_DIS
LIN {X -103.204,Y -19.551,Z -35.794,A -90.000,B 90.000,C 0.000} C_DIS
LIN {X -103.025,Y -19.536,Z -35.600,A -90.000,B 90.000,C 0.000} C_DIS
LIN {X -102.965,Y -19.533,Z -35.539,A -90.000,B 90.000,C 0.000} C_DIS
LIN {X -102.812,Y -19.520,Z -35.398,A -90.000,B 90.000,C 0.000} C_DIS
LIN {X -102.463,Y -19.497,Z -35.099,A -90.000,B 90.000,C 0.000} C_DIS
LIN {X -102.328,Y -19.489,Z -34.987,A -90.000,B 90.000,C 0.000} C_DIS
LIN {X -102.179,Y -19.482,Z -34.867,A -90.000,B 90.000,C 0.000} C_DIS
LIN {X -101.857,Y -19.455,Z -34.617,A -90.000,B 90.000,C 0.000} C_DIS
LIN {X -101.679,Y -19.444,Z -34.486,A -90.000,B 90.000,C 0.000} C_DIS
LIN {X -101.386,Y -19.427,Z -34.285,A -90.000,B 90.000,C 0.000} C_DIS
LIN {X -101.162,Y -19.412,Z -34.133,A -90.000,B 90.000,C 0.000} C_DIS
LIN {X -100.839,Y -19.397,Z -33.929,A -90.000,B 90.000,C 0.000} C_DIS
LIN {X -100.098,Y -19.374,Z -33.487,A -90.000,B 90.000,C 0.000} C_DIS
LIN {X -99.759,Y -19.363,Z -33.289,A -90.000,B 90.000,C 0.000} C_DIS
LIN {X -99.092,Y -19.344,Z -32.925,A -90.000,B 90.000,C 0.000} C_DIS
LIN {X -98.838,Y -19.336,Z -32.796,A -90.000,B 90.000,C 0.000} C_DIS
LIN {X -98.570,Y -19.322,Z -32.645,A -90.000,B 90.000,C 0.000} C_DIS
LIN {X -98.379,Y -19.311,Z -32.544,A -90.000,B 90.000,C 0.000} C_DIS
LIN {X -98.345,Y -19.310,Z -32.526,A -90.000,B 90.000,C 0.000} C_DIS
LIN {X -98.344,Y -19.308,Z -32.523,A -90.000,B 90.000,C 0.000} C_DIS
LIN {X -98.344,Y -60.000,Z -32.523,A -90.000,B 90.000,C 0.000} C_DIS
LIN {X -108.493,Y -60.000,Z -243.561,A -90.000,B 90.000,C 0.000} C_DIS
LIN {X -108.493,Y -19.308,Z -243.561,A -90.000,B 90.000,C 0.000} C_DIS
LIN {X -107.711,Y -19.308,Z -243.031,A -90.000,B 90.000,C 0.000} C_DIS
LIN {X -106.239,Y -19.308,Z -242.009,A -90.000,B 90.000,C 0.000} C_DIS
LIN {X -100.134,Y -19.308,Z -237.742,A -90.000,B 90.000,C 0.000} C_DIS
LIN {X -96.953,Y -19.308,Z -235.513,A -90.000,B 90.000,C 0.000} C_DIS
LIN {X -93.878,Y -19.308,Z -233.382,A -90.000,B 90.000,C 0.000} C_DIS
LIN {X -88.767,Y -19.308,Z -229.837,A -90.000,B 90.000,C 0.000} C_DIS
LIN {X -87.200,Y -19.308,Z -228.775,A -90.000,B 90.000,C 0.000} C_DIS
LIN {X -80.694,Y -19.308,Z -224.348,A -90.000,B 90.000,C 0.000} C_DIS
LIN {X -72.537,Y -19.308,Z -218.944,A -90.000,B 90.000,C 0.000} C_DIS
LIN {X -69.953,Y -19.308,Z -217.240,A -90.000,B 90.000,C 0.000} C_DIS
LIN {X -64.534,Y -19.308,Z -213.689,A -90.000,B 90.000,C 0.000} C_DIS
LIN {X -59.643,Y -19.308,Z -210.435,A -90.000,B 90.000,C 0.000} C_DIS
LIN {X -57.077,Y -19.308,Z -208.741,A -90.000,B 90.000,C 0.000} C_DIS
LIN {X -50.717,Y -19.308,Z -204.386,A -90.000,B 90.000,C 0.000} C_DIS
LIN {X -45.269,Y -19.308,Z -200.522,A -90.000,B 90.000,C 0.000} C_DIS
LIN {X -40.819,Y -19.308,Z -197.200,A -90.000,B 90.000,C 0.000} C_DIS
LIN {X -39.920,Y -19.308,Z -196.511,A -90.000,B 90.000,C 0.000} C_DIS
LIN {X -37.026,Y -19.308,Z -194.251,A -90.000,B 90.000,C 0.000} C_DIS
LIN {X -35.719,Y -19.308,Z -193.226,A -90.000,B 90.000,C 0.000} C_DIS
LIN {X -32.079,Y -19.308,Z -190.305,A -90.000,B 90.000,C 0.000} C_DIS
LIN {X -30.580,Y -19.308,Z -189.131,A -90.000,B 90.000,C 0.000} C_DIS
LIN {X -29.126,Y -19.308,Z -187.938,A -90.000,B 90.000,C 0.000} C_DIS
LIN {X -27.667,Y -19.308,Z -186.768,A -90.000,B 90.000,C 0.000} C_DIS
LIN {X -26.278,Y -19.308,Z -185.572,A -90.000,B 90.000,C 0.000} C_DIS
LIN {X -25.065,Y -19.308,Z -184.554,A -90.000,B 90.000,C 0.000} C_DIS
LIN {X -23.871,Y -19.308,Z -183.449,A -90.000,B 90.000,C 0.000} C_DIS
LIN {X -22.618,Y -19.308,Z -182.321,A -90.000,B 90.000,C 0.000} C_DIS
LIN {X -21.630,Y -19.308,Z -181.351,A -90.000,B 90.000,C 0.000} C_DIS
LIN {X -20.081,Y -19.308,Z -179.786,A -90.000,B 90.000,C 0.000} C_DIS
LIN {X -19.428,Y -19.308,Z -179.081,A -90.000,B 90.000,C 0.000} C_DIS
LIN {X -17.894,Y -19.308,Z -177.372,A -90.000,B 90.000,C 0.000} C_DIS
LIN {X -17.343,Y -19.308,Z -176.711,A -90.000,B 90.000,C 0.000} C_DIS
LIN {X -15.783,Y -19.308,Z -174.767,A -90.000,B 90.000,C 0.000} C_DIS
LIN {X -15.202,Y -19.308,Z -173.982,A -90.000,B 90.000,C 0.000} C_DIS
LIN {X -13.976,Y -19.308,Z -172.233,A -90.000,B 90.000,C 0.000} C_DIS
LIN {X -13.565,Y -19.308,Z -171.593,A -90.000,B 90.000,C 0.000} C_DIS
LIN {X -12.251,Y -19.308,Z -169.374,A -90.000,B 90.000,C 0.000} C_DIS
LIN {X -12.164,Y -19.308,Z -169.209,A -90.000,B 90.000,C 0.000} C_DIS
LIN {X -11.037,Y -19.308,Z -166.833,A -90.000,B 90.000,C 0.000} C_DIS
LIN {X -10.270,Y -19.308,Z -164.568,A -90.000,B 90.000,C 0.000} C_DIS
LIN {X -9.988,Y -19.308,Z -162.844,A -90.000,B 90.000,C 0.000} C_DIS
LIN {X -10.094,Y -19.308,Z -161.837,A -90.000,B 90.000,C 0.000} C_DIS
LIN {X -10.396,Y -19.308,Z -161.101,A -90.000,B 90.000,C 0.000} C_DIS
LIN {X -10.414,Y -19.308,Z -161.047,A -90.000,B 90.000,C 0.000} C_DIS
LIN {X -10.692,Y -19.308,Z -160.659,A -90.000,B 90.000,C 0.000} C_DIS
LIN {X -10.931,Y -19.308,Z -160.280,A -90.000,B 90.000,C 0.000} C_DIS
LIN {X -11.437,Y -19.308,Z -159.744,A -90.000,B 90.000,C 0.000} C_DIS
LIN {X -11.945,Y -19.308,Z -159.133,A -90.000,B 90.000,C 0.000} C_DIS
LIN {X -12.566,Y -19.308,Z -158.450,A -90.000,B 90.000,C 0.000} C_DIS
LIN {X -12.843,Y -19.308,Z -158.174,A -90.000,B 90.000,C 0.000} C_DIS
LIN {X -13.827,Y -19.308,Z -157.168,A -90.000,B 90.000,C 0.000} C_DIS
LIN {X -14.224,Y -19.308,Z -156.797,A -90.000,B 90.000,C 0.000} C_DIS
LIN {X -15.554,Y -19.308,Z -155.525,A -90.000,B 90.000,C 0.000} C_DIS
LIN {X -16.006,Y -19.308,Z -155.122,A -90.000,B 90.000,C 0.000} C_DIS
LIN {X -17.865,Y -19.308,Z -153.434,A -90.000,B 90.000,C 0.000} C_DIS
LIN {X -18.271,Y -19.308,Z -153.081,A -90.000,B 90.000,C 0.000} C_DIS
LIN {X -20.739,Y -19.308,Z -150.918,A -90.000,B 90.000,C 0.000} C_DIS
LIN {X -21.160,Y -19.308,Z -150.558,A -90.000,B 90.000,C 0.000} C_DIS
LIN {X -23.600,Y -19.308,Z -148.316,A -90.000,B 90.000,C 0.000} C_DIS
LIN {X -24.337,Y -19.308,Z -147.648,A -90.000,B 90.000,C 0.000} C_DIS
LIN {X -24.655,Y -19.308,Z -147.336,A -90.000,B 90.000,C 0.000} C_DIS
LIN {X -26.684,Y -19.308,Z -145.263,A -90.000,B 90.000,C 0.000} C_DIS
LIN {X -27.934,Y -19.308,Z -143.998,A -90.000,B 90.000,C 0.000} C_DIS
LIN {X -29.542,Y -19.308,Z -142.048,A -90.000,B 90.000,C 0.000} C_DIS
LIN {X -31.140,Y -19.308,Z -140.122,A -90.000,B 90.000,C 0.000} C_DIS
LIN {X -31.270,Y -19.308,Z -139.964,A -90.000,B 90.000,C 0.000} C_DIS
LIN {X -31.533,Y -19.308,Z -139.567,A -90.000,B 90.000,C 0.000} C_DIS
LIN {X -33.416,Y -19.308,Z -136.599,A -90.000,B 90.000,C 0.000} C_DIS
LIN {X -34.032,Y -19.308,Z -135.623,A -90.000,B 90.000,C 0.000} C_DIS
LIN {X -34.252,Y -19.308,Z -135.201,A -90.000,B 90.000,C 0.000} C_DIS
LIN {X -35.633,Y -19.308,Z -132.517,A -90.000,B 90.000,C 0.000} C_DIS
LIN {X -36.275,Y -19.308,Z -131.244,A -90.000,B 90.000,C 0.000} C_DIS
LIN {X -36.634,Y -19.308,Z -130.433,A -90.000,B 90.000,C 0.000} C_DIS
LIN {X -37.897,Y -19.308,Z -127.529,A -90.000,B 90.000,C 0.000} C_DIS
LIN {X -39.071,Y -19.308,Z -124.706,A -90.000,B 90.000,C 0.000} C_DIS
LIN {X -39.217,Y -19.308,Z -124.347,A -90.000,B 90.000,C 0.000} C_DIS
LIN {X -39.321,Y -19.308,Z -124.112,A -90.000,B 90.000,C 0.000} C_DIS
LIN {X -39.784,Y -19.308,Z -123.087,A -90.000,B 90.000,C 0.000} C_DIS
LIN {X -40.230,Y -19.308,Z -122.175,A -90.000,B 90.000,C 0.000} C_DIS
LIN {X -40.527,Y -19.308,Z -121.611,A -90.000,B 90.000,C 0.000} C_DIS
LIN {X -41.107,Y -19.308,Z -120.577,A -90.000,B 90.000,C 0.000} C_DIS
LIN {X -41.216,Y -19.308,Z -120.411,A -90.000,B 90.000,C 0.000} C_DIS
LIN {X -42.087,Y -19.308,Z -119.102,A -90.000,B 90.000,C 0.000} C_DIS
LIN {X -43.095,Y -19.308,Z -117.765,A -90.000,B 90.000,C 0.000} C_DIS
LIN {X -43.291,Y -19.308,Z -117.501,A -90.000,B 90.000,C 0.000} C_DIS
LIN {X -43.743,Y -19.308,Z -116.923,A -90.000,B 90.000,C 0.000} C_DIS
LIN {X -46.833,Y -19.308,Z -113.018,A -90.000,B 90.000,C 0.000} C_DIS
LIN {X -47.614,Y -19.308,Z -112.037,A -90.000,B 90.000,C 0.000} C_DIS
LIN {X -50.081,Y -19.308,Z -108.890,A -90.000,B 90.000,C 0.000} C_DIS
LIN {X -50.816,Y -19.308,Z -107.929,A -90.000,B 90.000,C 0.000} C_DIS
LIN {X -52.043,Y -19.308,Z -106.310,A -90.000,B 90.000,C 0.000} C_DIS
LIN {X -52.680,Y -19.308,Z -105.480,A -90.000,B 90.000,C 0.000} C_DIS
LIN {X -53.697,Y -19.308,Z -104.091,A -90.000,B 90.000,C 0.000} C_DIS
LIN {X -55.259,Y -19.308,Z -102.003,A -90.000,B 90.000,C 0.000} C_DIS
LIN {X -56.679,Y -19.308,Z -100.064,A -90.000,B 90.000,C 0.000} C_DIS
LIN {X -57.644,Y -19.308,Z -98.785,A -90.000,B 90.000,C 0.000} C_DIS
LIN {X -57.760,Y -19.308,Z -98.630,A -90.000,B 90.000,C 0.000} C_DIS
LIN {X -57.957,Y -19.308,Z -98.370,A -90.000,B 90.000,C 0.000} C_DIS
LIN {X -59.971,Y -19.308,Z -95.692,A -90.000,B 90.000,C 0.000} C_DIS
LIN {X -60.783,Y -19.308,Z -94.631,A -90.000,B 90.000,C 0.000} C_DIS
LIN {X -62.098,Y -19.308,Z -92.954,A -90.000,B 90.000,C 0.000} C_DIS
LIN {X -62.264,Y -19.308,Z -92.748,A -90.000,B 90.000,C 0.000} C_DIS
LIN {X -62.726,Y -19.308,Z -92.183,A -90.000,B 90.000,C 0.000} C_DIS
LIN {X -63.970,Y -19.308,Z -90.639,A -90.000,B 90.000,C 0.000} C_DIS
LIN {X -65.421,Y -19.308,Z -88.928,A -90.000,B 90.000,C 0.000} C_DIS
LIN {X -65.598,Y -19.308,Z -88.723,A -90.000,B 90.000,C 0.000} C_DIS
LIN {X -67.351,Y -19.308,Z -86.782,A -90.000,B 90.000,C 0.000} C_DIS
LIN {X -68.228,Y -19.308,Z -85.873,A -90.000,B 90.000,C 0.000} C_DIS
LIN {X -69.116,Y -19.308,Z -84.929,A -90.000,B 90.000,C 0.000} C_DIS
LIN {X -70.889,Y -19.308,Z -83.113,A -90.000,B 90.000,C 0.000} C_DIS
LIN {X -72.212,Y -19.308,Z -81.817,A -90.000,B 90.000,C 0.000} C_DIS
LIN {X -72.479,Y -19.308,Z -81.570,A -90.000,B 90.000,C 0.000} C_DIS
LIN {X -73.903,Y -19.308,Z -80.302,A -90.000,B 90.000,C 0.000} C_DIS
LIN {X -74.794,Y -19.308,Z -79.651,A -90.000,B 90.000,C 0.000} C_DIS
LIN {X -74.950,Y -19.308,Z -79.545,A -90.000,B 90.000,C 0.000} C_DIS
LIN {X -76.029,Y -19.308,Z -79.054,A -90.000,B 90.000,C 0.000} C_DIS
LIN {X -77.301,Y -19.308,Z -78.674,A -90.000,B 90.000,C 0.000} C_DIS
LIN {X -77.888,Y -19.308,Z -78.513,A -90.000,B 90.000,C 0.000} C_DIS
LIN {X -78.650,Y -19.308,Z -78.279,A -90.000,B 90.000,C 0.000} C_DIS
LIN {X -79.052,Y -19.308,Z -78.132,A -90.000,B 90.000,C 0.000} C_DIS
LIN {X -80.625,Y -19.308,Z -77.543,A -90.000,B 90.000,C 0.000} C_DIS
LIN {X -80.768,Y -19.308,Z -77.479,A -90.000,B 90.000,C 0.000} C_DIS
LIN {X -81.195,Y -19.308,Z -77.267,A -90.000,B 90.000,C 0.000} C_DIS
LIN {X -81.583,Y -19.308,Z -77.051,A -90.000,B 90.000,C 0.000} C_DIS
LIN {X -82.777,Y -19.308,Z -76.396,A -90.000,B 90.000,C 0.000} C_DIS
LIN {X -83.199,Y -19.308,Z -76.129,A -90.000,B 90.000,C 0.000} C_DIS
LIN {X -83.508,Y -19.308,Z -75.927,A -90.000,B 90.000,C 0.000} C_DIS
LIN {X -84.763,Y -19.308,Z -75.057,A -90.000,B 90.000,C 0.000} C_DIS
LIN {X -85.185,Y -19.308,Z -74.743,A -90.000,B 90.000,C 0.000} C_DIS
LIN {X -85.424,Y -19.308,Z -74.565,A -90.000,B 90.000,C 0.000} C_DIS
LIN {X -85.681,Y -19.308,Z -74.367,A -90.000,B 90.000,C 0.000} C_DIS
LIN {X -85.829,Y -19.308,Z -74.262,A -90.000,B 90.000,C 0.000} C_DIS
LIN {X -85.978,Y -19.308,Z -74.151,A -90.000,B 90.000,C 0.000} C_DIS
LIN {X -86.147,Y -19.308,Z -74.021,A -90.000,B 90.000,C 0.000} C_DIS
LIN {X -86.531,Y -19.308,Z -73.755,A -90.000,B 90.000,C 0.000} C_DIS
LIN {X -86.813,Y -19.308,Z -73.554,A -90.000,B 90.000,C 0.000} C_DIS
LIN {X -87.534,Y -19.308,Z -73.015,A -90.000,B 90.000,C 0.000} C_DIS
LIN {X -87.774,Y -19.308,Z -72.821,A -90.000,B 90.000,C 0.000} C_DIS
LIN {X -88.166,Y -19.308,Z -72.500,A -90.000,B 90.000,C 0.000} C_DIS
LIN {X -88.246,Y -19.308,Z -72.438,A -90.000,B 90.000,C 0.000} C_DIS
LIN {X -88.675,Y -19.308,Z -72.089,A -90.000,B 90.000,C 0.000} C_DIS
LIN {X -89.349,Y -19.308,Z -71.487,A -90.000,B 90.000,C 0.000} C_DIS
LIN {X -89.440,Y -19.308,Z -71.403,A -90.000,B 90.000,C 0.000} C_DIS
LIN {X -90.026,Y -19.308,Z -70.837,A -90.000,B 90.000,C 0.000} C_DIS
LIN {X -90.361,Y -19.308,Z -70.524,A -90.000,B 90.000,C 0.000} C_DIS
LIN {X -90.673,Y -19.308,Z -70.218,A -90.000,B 90.000,C 0.000} C_DIS
LIN {X -91.040,Y -19.308,Z -69.899,A -90.000,B 90.000,C 0.000} C_DIS
LIN {X -91.249,Y -19.308,Z -69.704,A -90.000,B 90.000,C 0.000} C_DIS
LIN {X -91.444,Y -19.308,Z -69.552,A -90.000,B 90.000,C 0.000} C_DIS
LIN {X -91.733,Y -19.308,Z -69.314,A -90.000,B 90.000,C 0.000} C_DIS
LIN {X -91.780,Y -19.308,Z -69.282,A -90.000,B 90.000,C 0.000} C_DIS
LIN {X -92.439,Y -19.308,Z -68.807,A -90.000,B 90.000,C 0.000} C_DIS
LIN {X -92.718,Y -19.308,Z -68.616,A -90.000,B 90.000,C 0.000} C_DIS
LIN {X -93.286,Y -19.308,Z -68.215,A -90.000,B 90.000,C 0.000} C_DIS
LIN {X -93.825,Y -19.308,Z -67.855,A -90.000,B 90.000,C 0.000} C_DIS
LIN {X -94.769,Y -19.308,Z -67.164,A -90.000,B 90.000,C 0.000} C_DIS
LIN {X -95.022,Y -19.308,Z -66.962,A -90.000,B 90.000,C 0.000} C_DIS
LIN {X -95.711,Y -19.308,Z -66.425,A -90.000,B 90.000,C 0.000} C_DIS
LIN {X -96.155,Y -19.308,Z -66.059,A -90.000,B 90.000,C 0.000} C_DIS
LIN {X -96.219,Y -19.308,Z -66.011,A -90.000,B 90.000,C 0.000} C_DIS
LIN {X -97.029,Y -19.308,Z -65.356,A -90.000,B 90.000,C 0.000} C_DIS
LIN {X -97.202,Y -19.308,Z -65.221,A -90.000,B 90.000,C 0.000} C_DIS
LIN {X -98.120,Y -19.308,Z -64.471,A -90.000,B 90.000,C 0.000} C_DIS
LIN {X -99.212,Y -19.308,Z -63.589,A -90.000,B 90.000,C 0.000} C_DIS
LIN {X -99.812,Y -19.308,Z -63.119,A -90.000,B 90.000,C 0.000} C_DIS
LIN {X -100.608,Y -19.308,Z -62.479,A -90.000,B 90.000,C 0.000} C_DIS
LIN {X -101.011,Y -19.308,Z -62.175,A -90.000,B 90.000,C 0.000} C_DIS
LIN {X -101.441,Y -19.308,Z -61.844,A -90.000,B 90.000,C 0.000} C_DIS
LIN {X -101.817,Y -19.308,Z -61.547,A -90.000,B 90.000,C 0.000} C_DIS
LIN {X -102.389,Y -19.308,Z -61.107,A -90.000,B 90.000,C 0.000} C_DIS
LIN {X -102.735,Y -19.308,Z -60.811,A -90.000,B 90.000,C 0.000} C_DIS
LIN {X -103.121,Y -19.308,Z -60.467,A -90.000,B 90.000,C 0.000} C_DIS
LIN {X -103.650,Y -19.308,Z -60.012,A -90.000,B 90.000,C 0.000} C_DIS
LIN {X -103.689,Y -19.308,Z -59.974,A -90.000,B 90.000,C 0.000} C_DIS
LIN {X -104.099,Y -19.308,Z -59.552,A -90.000,B 90.000,C 0.000} C_DIS
LIN {X -104.421,Y -19.308,Z -59.235,A -90.000,B 90.000,C 0.000} C_DIS
LIN {X -104.733,Y -19.308,Z -58.903,A -90.000,B 90.000,C 0.000} C_DIS
LIN {X -104.832,Y -19.308,Z -58.791,A -90.000,B 90.000,C 0.000} C_DIS
LIN {X -104.955,Y -19.308,Z -58.658,A -90.000,B 90.000,C 0.000} C_DIS
LIN {X -105.376,Y -19.308,Z -58.161,A -90.000,B 90.000,C 0.000} C_DIS
LIN {X -105.696,Y -19.308,Z -57.742,A -90.000,B 90.000,C 0.000} C_DIS
LIN {X -105.930,Y -19.308,Z -57.430,A -90.000,B 90.000,C 0.000} C_DIS
LIN {X -106.038,Y -19.308,Z -57.285,A -90.000,B 90.000,C 0.000} C_DIS
LIN {X -106.208,Y -19.308,Z -57.065,A -90.000,B 90.000,C 0.000} C_DIS
LIN {X -106.425,Y -19.308,Z -56.753,A -90.000,B 90.000,C 0.000} C_DIS
LIN {X -106.852,Y -19.308,Z -56.042,A -90.000,B 90.000,C 0.000} C_DIS
LIN {X -106.960,Y -19.308,Z -55.831,A -90.000,B 90.000,C 0.000} C_DIS
LIN {X -107.148,Y -19.308,Z -55.451,A -90.000,B 90.000,C 0.000} C_DIS
LIN {X -107.384,Y -19.308,Z -54.959,A -90.000,B 90.000,C 0.000} C_DIS
LIN {X -107.458,Y -19.308,Z -54.792,A -90.000,B 90.000,C 0.000} C_DIS
LIN {X -107.707,Y -19.308,Z -54.084,A -90.000,B 90.000,C 0.000} C_DIS
LIN {X -107.829,Y -19.308,Z -53.652,A -90.000,B 90.000,C 0.000} C_DIS
LIN {X -107.908,Y -19.308,Z -53.349,A -90.000,B 90.000,C 0.000} C_DIS
LIN {X -108.016,Y -19.308,Z -52.960,A -90.000,B 90.000,C 0.000} C_DIS
LIN {X -108.133,Y -19.308,Z -52.307,A -90.000,B 90.000,C 0.000} C_DIS
LIN {X -108.192,Y -19.308,Z -51.924,A -90.000,B 90.000,C 0.000} C_DIS
LIN {X -108.229,Y -19.308,Z -51.662,A -90.000,B 90.000,C 0.000} C_DIS
LIN {X -108.263,Y -19.308,Z -51.284,A -90.000,B 90.000,C 0.000} C_DIS
LIN {X -108.266,Y -19.308,Z -51.167,A -90.000,B 90.000,C 0.000} C_DIS
LIN {X -108.268,Y -19.308,Z -50.997,A -90.000,B 90.000,C 0.000} C_DIS
LIN {X -108.263,Y -19.308,Z -50.788,A -90.000,B 90.000,C 0.000} C_DIS
LIN {X -108.246,Y -19.308,Z -50.409,A -90.000,B 90.000,C 0.000} C_DIS
LIN {X -108.237,Y -19.308,Z -50.276,A -90.000,B 90.000,C 0.000} C_DIS
LIN {X -108.132,Y -19.308,Z -49.675,A -90.000,B 90.000,C 0.000} C_DIS
LIN {X -108.071,Y -19.308,Z -49.388,A -90.000,B 90.000,C 0.000} C_DIS
LIN {X -107.956,Y -19.308,Z -49.027,A -90.000,B 90.000,C 0.000} C_DIS
LIN {X -107.865,Y -19.308,Z -48.793,A -90.000,B 90.000,C 0.000} C_DIS
LIN {X -107.642,Y -19.308,Z -48.318,A -90.000,B 90.000,C 0.000} C_DIS
LIN {X -107.522,Y -19.308,Z -48.131,A -90.000,B 90.000,C 0.000} C_DIS
LIN {X -107.574,Y -19.308,Z -48.045,A -90.000,B 90.000,C 0.000} C_DIS
LIN {X -107.742,Y -19.308,Z -47.762,A -90.000,B 90.000,C 0.000} C_DIS
LIN {X -107.951,Y -19.308,Z -47.376,A -90.000,B 90.000,C 0.000} C_DIS
LIN {X -108.219,Y -19.308,Z -46.863,A -90.000,B 90.000,C 0.000} C_DIS
LIN {X -108.402,Y -19.308,Z -46.462,A -90.000,B 90.000,C 0.000} C_DIS
LIN {X -108.609,Y -19.308,Z -45.991,A -90.000,B 90.000,C 0.000} C_DIS
LIN {X -108.746,Y -19.308,Z -45.658,A -90.000,B 90.000,C 0.000} C_DIS
LIN {X -108.858,Y -19.308,Z -45.343,A -90.000,B 90.000,C 0.000} C_DIS
LIN {X -108.913,Y -19.308,Z -45.173,A -90.000,B 90.000,C 0.000} C_DIS
LIN {X -109.037,Y -19.308,Z -44.749,A -90.000,B 90.000,C 0.000} C_DIS
LIN {X -109.131,Y -19.308,Z -44.336,A -90.000,B 90.000,C 0.000} C_DIS
LIN {X -109.207,Y -19.308,Z -43.946,A -90.000,B 90.000,C 0.000} C_DIS
LIN {X -109.299,Y -19.308,Z -43.285,A -90.000,B 90.000,C 0.000} C_DIS
LIN {X -109.329,Y -19.308,Z -42.928,A -90.000,B 90.000,C 0.000} C_DIS
LIN {X -109.338,Y -19.308,Z -42.525,A -90.000,B 90.000,C 0.000} C_DIS
LIN {X -109.325,Y -19.308,Z -42.194,A -90.000,B 90.000,C 0.000} C_DIS
LIN {X -109.300,Y -19.308,Z -41.834,A -90.000,B 90.000,C 0.000} C_DIS
LIN {X -109.289,Y -19.308,Z -41.728,A -90.000,B 90.000,C 0.000} C_DIS
LIN {X -109.240,Y -19.308,Z -41.427,A -90.000,B 90.000,C 0.000} C_DIS
LIN {X -109.168,Y -19.308,Z -41.028,A -90.000,B 90.000,C 0.000} C_DIS
LIN {X -109.086,Y -19.308,Z -40.740,A -90.000,B 90.000,C 0.000} C_DIS
LIN {X -108.962,Y -19.308,Z -40.353,A -90.000,B 90.000,C 0.000} C_DIS
LIN {X -108.854,Y -19.308,Z -40.085,A -90.000,B 90.000,C 0.000} C_DIS
LIN {X -108.693,Y -19.308,Z -39.742,A -90.000,B 90.000,C 0.000} C_DIS
LIN {X -108.563,Y -19.308,Z -39.488,A -90.000,B 90.000,C 0.000} C_DIS
LIN {X -108.358,Y -19.308,Z -39.169,A -90.000,B 90.000,C 0.000} C_DIS
LIN {X -108.164,Y -19.308,Z -38.902,A -90.000,B 90.000,C 0.000} C_DIS
LIN {X -107.954,Y -19.308,Z -38.653,A -90.000,B 90.000,C 0.000} C_DIS
LIN {X -107.734,Y -19.308,Z -38.449,A -90.000,B 90.000,C 0.000} C_DIS
LIN {X -107.485,Y -19.308,Z -38.221,A -90.000,B 90.000,C 0.000} C_DIS
LIN {X -107.350,Y -19.308,Z -38.122,A -90.000,B 90.000,C 0.000} C_DIS
LIN {X -107.187,Y -19.308,Z -38.009,A -90.000,B 90.000,C 0.000} C_DIS
LIN {X -107.101,Y -19.308,Z -37.954,A -90.000,B 90.000,C 0.000} C_DIS
LIN {X -106.954,Y -19.308,Z -37.879,A -90.000,B 90.000,C 0.000} C_DIS
LIN {X -106.772,Y -19.308,Z -37.781,A -90.000,B 90.000,C 0.000} C_DIS
LIN {X -106.437,Y -19.308,Z -37.609,A -90.000,B 90.000,C 0.000} C_DIS
LIN {X -106.079,Y -19.308,Z -37.483,A -90.000,B 90.000,C 0.000} C_DIS
LIN {X -105.826,Y -19.308,Z -37.408,A -90.000,B 90.000,C 0.000} C_DIS
LIN {X -105.429,Y -19.308,Z -37.317,A -90.000,B 90.000,C 0.000} C_DIS
LIN {X -105.058,Y -19.308,Z -37.239,A -90.000,B 90.000,C 0.000} C_DIS
LIN {X -105.035,Y -19.308,Z -37.208,A -90.000,B 90.000,C 0.000} C_DIS
LIN {X -104.718,Y -19.308,Z -36.757,A -90.000,B 90.000,C 0.000} C_DIS
LIN {X -104.582,Y -19.308,Z -36.579,A -90.000,B 90.000,C 0.000} C_DIS
LIN {X -104.232,Y -19.308,Z -36.145,A -90.000,B 90.000,C 0.000} C_DIS
LIN {X -104.094,Y -19.308,Z -35.987,A -90.000,B 90.000,C 0.000} C_DIS
LIN {X -104.008,Y -19.308,Z -35.903,A -90.000,B 90.000,C 0.000} C_DIS
LIN {X -103.742,Y -19.308,Z -35.667,A -90.000,B 90.000,C 0.000} C_DIS
LIN {X -103.347,Y -19.308,Z -35.321,A -90.000,B 90.000,C 0.000} C_DIS
LIN {X -103.063,Y -19.308,Z -35.113,A -90.000,B 90.000,C 0.000} C_DIS
LIN {X -102.475,Y -19.308,Z -34.699,A -90.000,B 90.000,C 0.000} C_DIS
LIN {X -101.853,Y -19.308,Z -34.319,A -90.000,B 90.000,C 0.000} C_DIS
LIN {X -101.153,Y -19.308,Z -33.923,A -90.000,B 90.000,C 0.000} C_DIS
LIN {X -100.339,Y -19.308,Z -33.484,A -90.000,B 90.000,C 0.000} C_DIS
LIN {X -99.768,Y -19.308,Z -33.186,A -90.000,B 90.000,C 0.000} C_DIS
LIN {X -99.192,Y -19.308,Z -32.905,A -90.000,B 90.000,C 0.000} C_DIS
LIN {X -99.016,Y -19.308,Z -32.828,A -90.000,B 90.000,C 0.000} C_DIS
LIN {X -98.595,Y -19.308,Z -32.632,A -90.000,B 90.000,C 0.000} C_DIS
LIN {X -98.149,Y -19.308,Z -32.439,A -90.000,B 90.000,C 0.000} C_DIS
LIN {X -98.151,Y -19.308,Z -32.383,A -90.000,B 90.000,C 0.000} C_DIS
LIN {X -98.158,Y -19.308,Z -32.263,A -90.000,B 90.000,C 0.000} C_DIS
LIN {X -98.147,Y -19.308,Z -31.940,A -90.000,B 90.000,C 0.000} C_DIS
LIN {X -98.124,Y -19.308,Z -31.669,A -90.000,B 90.000,C 0.000} C_DIS
LIN {X -98.109,Y -19.308,Z -31.585,A -90.000,B 90.000,C 0.000} C_DIS
LIN {X -98.048,Y -19.308,Z -31.319,A -90.000,B 90.000,C 0.000} C_DIS
LIN {X -98.023,Y -19.308,Z -31.238,A -90.000,B 90.000,C 0.000} C_DIS
LIN {X -97.846,Y -19.308,Z -30.724,A -90.000,B 90.000,C 0.000} C_DIS
LIN {X -97.798,Y -19.308,Z -30.599,A -90.000,B 90.000,C 0.000} C_DIS
LIN {X -97.736,Y -19.308,Z -30.462,A -90.000,B 90.000,C 0.000} C_DIS
LIN {X -97.698,Y -19.308,Z -30.386,A -90.000,B 90.000,C 0.000} C_DIS
LIN {X -97.405,Y -19.308,Z -29.838,A -90.000,B 90.000,C 0.000} C_DIS
LIN {X -97.309,Y -19.308,Z -29.685,A -90.000,B 90.000,C 0.000} C_DIS
LIN {X -96.912,Y -19.308,Z -29.089,A -90.000,B 90.000,C 0.000} C_DIS
LIN {X -96.612,Y -19.308,Z -28.693,A -90.000,B 90.000,C 0.000} C_DIS
LIN {X -96.351,Y -19.308,Z -28.374,A -90.000,B 90.000,C 0.000} C_DIS
LIN {X -96.104,Y -19.308,Z -28.082,A -90.000,B 90.000,C 0.000} C_DIS
LIN {X -95.874,Y -19.308,Z -27.826,A -90.000,B 90.000,C 0.000} C_DIS
LIN {X -95.659,Y -19.308,Z -27.611,A -90.000,B 90.000,C 0.000} C_DIS
LIN {X -95.225,Y -19.308,Z -27.218,A -90.000,B 90.000,C 0.000} C_DIS
LIN {X -95.068,Y -19.308,Z -27.087,A -90.000,B 90.000,C 0.000} C_DIS
LIN {X -94.968,Y -19.308,Z -27.013,A -90.000,B 90.000,C 0.000} C_DIS
LIN {X -94.767,Y -19.308,Z -26.874,A -90.000,B 90.000,C 0.000} C_DIS
LIN {X -94.665,Y -19.308,Z -26.809,A -90.000,B 90.000,C 0.000} C_DIS
LIN {X -94.602,Y -19.308,Z -26.774,A -90.000,B 90.000,C 0.000} C_DIS
LIN {X -94.457,Y -19.308,Z -26.686,A -90.000,B 90.000,C 0.000} C_DIS
LIN {X -94.119,Y -19.308,Z -26.514,A -90.000,B 90.000,C 0.000} C_DIS
LIN {X -93.762,Y -19.308,Z -26.387,A -90.000,B 90.000,C 0.000} C_DIS
LIN {X -93.535,Y -19.308,Z -26.309,A -90.000,B 90.000,C 0.000} C_DIS
LIN {X -93.202,Y -19.308,Z -26.207,A -90.000,B 90.000,C 0.000} C_DIS
LIN {X -93.091,Y -19.308,Z -26.175,A -90.000,B 90.000,C 0.000} C_DIS
LIN {X -92.698,Y -19.308,Z -26.084,A -90.000,B 90.000,C 0.000} C_DIS
LIN {X -92.440,Y -19.308,Z -26.041,A -90.000,B 90.000,C 0.000} C_DIS
LIN {X -92.055,Y -19.308,Z -25.956,A -90.000,B 90.000,C 0.000} C_DIS
LIN {X -91.962,Y -19.308,Z -25.940,A -90.000,B 90.000,C 0.000} C_DIS
LIN {X -91.684,Y -19.308,Z -25.896,A -90.000,B 90.000,C 0.000} C_DIS
LIN {X -91.238,Y -19.308,Z -25.811,A -90.000,B 90.000,C 0.000} C_DIS
LIN {X -90.914,Y -19.308,Z -25.732,A -90.000,B 90.000,C 0.000} C_DIS
LIN {X -90.791,Y -19.308,Z -25.705,A -90.000,B 90.000,C 0.000} C_DIS
LIN {X -90.557,Y -19.308,Z -25.655,A -90.000,B 90.000,C 0.000} C_DIS
LIN {X -90.382,Y -19.308,Z -25.599,A -90.000,B 90.000,C 0.000} C_DIS
LIN {X -89.918,Y -19.308,Z -25.466,A -90.000,B 90.000,C 0.000} C_DIS
LIN {X -89.584,Y -19.308,Z -25.346,A -90.000,B 90.000,C 0.000} C_DIS
LIN {X -89.138,Y -19.308,Z -25.161,A -90.000,B 90.000,C 0.000} C_DIS
LIN {X -89.004,Y -19.308,Z -25.110,A -90.000,B 90.000,C 0.000} C_DIS
LIN {X -88.522,Y -19.308,Z -24.887,A -90.000,B 90.000,C 0.000} C_DIS
LIN {X -88.205,Y -19.308,Z -24.724,A -90.000,B 90.000,C 0.000} C_DIS
LIN {X -88.055,Y -19.308,Z -24.652,A -90.000,B 90.000,C 0.000} C_DIS
LIN {X -87.608,Y -19.308,Z -24.396,A -90.000,B 90.000,C 0.000} C_DIS
LIN {X -87.096,Y -19.308,Z -24.049,A -90.000,B 90.000,C 0.000} C_DIS
LIN {X -86.872,Y -19.308,Z -23.877,A -90.000,B 90.000,C 0.000} C_DIS
LIN {X -86.565,Y -19.308,Z -23.582,A -90.000,B 90.000,C 0.000} C_DIS
LIN {X -86.256,Y -19.308,Z -23.233,A -90.000,B 90.000,C 0.000} C_DIS
LIN {X -85.933,Y -19.308,Z -22.817,A -90.000,B 90.000,C 0.000} C_DIS
LIN {X -85.775,Y -19.308,Z -22.601,A -90.000,B 90.000,C 0.000} C_DIS
LIN {X -85.413,Y -19.308,Z -22.122,A -90.000,B 90.000,C 0.000} C_DIS
LIN {X -85.112,Y -19.308,Z -21.726,A -90.000,B 90.000,C 0.000} C_DIS
LIN {X -84.977,Y -19.308,Z -21.543,A -90.000,B 90.000,C 0.000} C_DIS
LIN {X -84.806,Y -19.308,Z -21.324,A -90.000,B 90.000,C 0.000} C_DIS
LIN {X -84.593,Y -19.308,Z -21.041,A -90.000,B 90.000,C 0.000} C_DIS
LIN {X -84.466,Y -19.308,Z -20.846,A -90.000,B 90.000,C 0.000} C_DIS
LIN {X -84.367,Y -19.308,Z -20.688,A -90.000,B 90.000,C 0.000} C_DIS
LIN {X -84.090,Y -19.308,Z -20.187,A -90.000,B 90.000,C 0.000} C_DIS
LIN {X -83.847,Y -19.308,Z -19.802,A -90.000,B 90.000,C 0.000} C_DIS
LIN {X -83.725,Y -19.308,Z -19.637,A -90.000,B 90.000,C 0.000} C_DIS
LIN {X -83.564,Y -19.308,Z -19.434,A -90.000,B 90.000,C 0.000} C_DIS
LIN {X -83.441,Y -19.308,Z -19.289,A -90.000,B 90.000,C 0.000} C_DIS
LIN {X -83.235,Y -19.308,Z -19.067,A -90.000,B 90.000,C 0.000} C_DIS
LIN {X -83.016,Y -19.308,Z -18.844,A -90.000,B 90.000,C 0.000} C_DIS
LIN {X -82.727,Y -19.308,Z -18.572,A -90.000,B 90.000,C 0.000} C_DIS
LIN {X -82.691,Y -19.308,Z -18.543,A -90.000,B 90.000,C 0.000} C_DIS
LIN {X -82.373,Y -19.308,Z -18.307,A -90.000,B 90.000,C 0.000} C_DIS
LIN {X -82.334,Y -19.308,Z -18.282,A -90.000,B 90.000,C 0.000} C_DIS
LIN {X -81.960,Y -19.308,Z -18.065,A -90.000,B 90.000,C 0.000} C_DIS
LIN {X -81.612,Y -19.308,Z -17.872,A -90.000,B 90.000,C 0.000} C_DIS
LIN {X -81.208,Y -19.308,Z -17.695,A -90.000,B 90.000,C 0.000} C_DIS
LIN {X -80.990,Y -19.308,Z -17.625,A -90.000,B 90.000,C 0.000} C_DIS
LIN {X -80.569,Y -19.308,Z -17.495,A -90.000,B 90.000,C 0.000} C_DIS
LIN {X -80.340,Y -19.308,Z -17.426,A -90.000,B 90.000,C 0.000} C_DIS
LIN {X -79.907,Y -19.308,Z -17.344,A -90.000,B 90.000,C 0.000} C_DIS
LIN {X -79.569,Y -19.308,Z -17.297,A -90.000,B 90.000,C 0.000} C_DIS
LIN {X -79.271,Y -19.308,Z -17.264,A -90.000,B 90.000,C 0.000} C_DIS
LIN {X -79.019,Y -19.308,Z -17.245,A -90.000,B 90.000,C 0.000} C_DIS
LIN {X -78.884,Y -19.308,Z -17.241,A -90.000,B 90.000,C 0.000} C_DIS
LIN {X -78.160,Y -19.308,Z -17.245,A -90.000,B 90.000,C 0.000} C_DIS
LIN {X -77.962,Y -19.308,Z -17.253,A -90.000,B 90.000,C 0.000} C_DIS
LIN {X -77.730,Y -19.308,Z -17.275,A -90.000,B 90.000,C 0.000} C_DIS
LIN {X -76.908,Y -19.308,Z -17.377,A -90.000,B 90.000,C 0.000} C_DIS
LIN {X -76.853,Y -19.308,Z -17.386,A -90.000,B 90.000,C 0.000} C_DIS
LIN {X -76.491,Y -19.308,Z -17.464,A -90.000,B 90.000,C 0.000} C_DIS
LIN {X -76.250,Y -19.308,Z -17.523,A -90.000,B 90.000,C 0.000} C_DIS
LIN {X -75.604,Y -19.308,Z -17.696,A -90.000,B 90.000,C 0.000} C_DIS
LIN {X -75.203,Y -19.308,Z -17.833,A -90.000,B 90.000,C 0.000} C_DIS
LIN {X -74.885,Y -19.308,Z -17.959,A -90.000,B 90.000,C 0.000} C_DIS
LIN {X -74.239,Y -19.308,Z -18.208,A -90.000,B 90.000,C 0.000} C_DIS
LIN {X -73.858,Y -19.308,Z -18.392,A -90.000,B 90.000,C 0.000} C_DIS
LIN {X -72.797,Y -19.308,Z -18.915,A -90.000,B 90.000,C 0.000} C_DIS
LIN {X -72.632,Y -19.308,Z -19.011,A -90.000,B 90.000,C 0.000} C_DIS
LIN {X -71.534,Y -19.308,Z -19.680,A -90.000,B 90.000,C 0.000} C_DIS
LIN {X -71.435,Y -19.308,Z -19.743,A -90.000,B 90.000,C 0.000} C_DIS
LIN {X -71.142,Y -19.308,Z -19.947,A -90.000,B 90.000,C 0.000} C_DIS
LIN {X -70.001,Y -19.308,Z -20.793,A -90.000,B 90.000,C 0.000} C_DIS
LIN {X -69.353,Y -19.308,Z -21.343,A -90.000,B 90.000,C 0.000} C_DIS
LIN {X -68.894,Y -19.308,Z -21.729,A -90.000,B 90.000,C 0.000} C_DIS
LIN {X -68.603,Y -19.308,Z -22.008,A -90.000,B 90.000,C 0.000} C_DIS
LIN {X -68.177,Y -19.308,Z -22.437,A -90.000,B 90.000,C 0.000} C_DIS
LIN {X -67.694,Y -19.308,Z -22.955,A -90.000,B 90.000,C 0.000} C_DIS
LIN {X -67.503,Y -19.308,Z -23.170,A -90.000,B 90.000,C 0.000} C_DIS
LIN {X -67.419,Y -19.308,Z -23.275,A -90.000,B 90.000,C 0.000} C_DIS
LIN {X -67.336,Y -19.308,Z -23.388,A -90.000,B 90.000,C 0.000} C_DIS
LIN {X -67.124,Y -19.308,Z -23.702,A -90.000,B 90.000,C 0.000} C_DIS
LIN {X -66.711,Y -19.308,Z -24.333,A -90.000,B 90.000,C 0.000} C_DIS
LIN {X -66.285,Y -19.308,Z -25.107,A -90.000,B 90.000,C 0.000} C_DIS
LIN {X -66.105,Y -19.308,Z -25.472,A -90.000,B 90.000,C 0.000} C_DIS
LIN {X -65.746,Y -19.308,Z -26.292,A -90.000,B 90.000,C 0.000} C_DIS
LIN {X -65.721,Y -19.308,Z -26.344,A -90.000,B 90.000,C 0.000} C_DIS
LIN {X -65.370,Y -19.308,Z -27.270,A -90.000,B 90.000,C 0.000} C_DIS
LIN {X -65.300,Y -19.308,Z -27.460,A -90.000,B 90.000,C 0.000} C_DIS
LIN {X -65.152,Y -19.308,Z -27.932,A -90.000,B 90.000,C 0.000} C_DIS
LIN {X -65.046,Y -19.308,Z -28.167,A -90.000,B 90.000,C 0.000} C_DIS
LIN {X -64.815,Y -19.308,Z -28.714,A -90.000,B 90.000,C 0.000} C_DIS
LIN {X -64.744,Y -19.308,Z -28.888,A -90.000,B 90.000,C 0.000} C_DIS
LIN {X -64.440,Y -19.308,Z -29.256,A -90.000,B 90.000,C 0.000} C_DIS
LIN {X -64.152,Y -19.308,Z -29.608,A -90.000,B 90.000,C 0.000} C_DIS
LIN {X -63.271,Y -19.308,Z -30.227,A -90.000,B 90.000,C 0.000} C_DIS
LIN {X -63.162,Y -19.308,Z -30.303,A -90.000,B 90.000,C 0.000} C_DIS
LIN {X -61.733,Y -19.308,Z -30.972,A -90.000,B 90.000,C 0.000} C_DIS
LIN {X -60.090,Y -19.308,Z -31.567,A -90.000,B 90.000,C 0.000} C_DIS
LIN {X -59.904,Y -19.308,Z -31.627,A -90.000,B 90.000,C 0.000} C_DIS
LIN {X -59.550,Y -19.308,Z -31.730,A -90.000,B 90.000,C 0.000} C_DIS
LIN {X -58.473,Y -19.308,Z -32.055,A -90.000,B 90.000,C 0.000} C_DIS
LIN {X -57.732,Y -19.308,Z -32.295,A -90.000,B 90.000,C 0.000} C_DIS
LIN {X -56.452,Y -19.308,Z -32.614,A -90.000,B 90.000,C 0.000} C_DIS
LIN {X -55.538,Y -19.308,Z -32.833,A -90.000,B 90.000,C 0.000} C_DIS
LIN {X -52.873,Y -19.308,Z -33.234,A -90.000,B 90.000,C 0.000} C_DIS
LIN {X -51.299,Y -19.308,Z -33.304,A -90.000,B 90.000,C 0.000} C_DIS
LIN {X -51.026,Y -19.308,Z -33.322,A -90.000,B 90.000,C 0.000} C_DIS
LIN {X -49.959,Y -19.308,Z -33.409,A -90.000,B 90.000,C 0.000} C_DIS
LIN {X -49.512,Y -19.308,Z -33.430,A -90.000,B 90.000,C 0.000} C_DIS
LIN {X -49.348,Y -19.308,Z -33.406,A -90.000,B 90.000,C 0.000} C_DIS
LIN {X -49.105,Y -19.308,Z -33.379,A -90.000,B 90.000,C 0.000} C_DIS
LIN {X -48.316,Y -19.308,Z -33.371,A -90.000,B 90.000,C 0.000} C_DIS
LIN {X -46.742,Y -19.308,Z -33.474,A -90.000,B 90.000,C 0.000} C_DIS
LIN {X -45.589,Y -19.308,Z -33.475,A -90.000,B 90.000,C 0.000} C_DIS
LIN {X -42.995,Y -19.308,Z -33.597,A -90.000,B 90.000,C 0.000} C_DIS
LIN {X -42.270,Y -19.308,Z -33.604,A -90.000,B 90.000,C 0.000} C_DIS
LIN {X -41.377,Y -19.308,Z -33.625,A -90.000,B 90.000,C 0.000} C_DIS
LIN {X -39.233,Y -19.308,Z -33.725,A -90.000,B 90.000,C 0.000} C_DIS
LIN {X -37.413,Y -19.308,Z -33.786,A -90.000,B 90.000,C 0.000} C_DIS
LIN {X -35.215,Y -19.308,Z -33.952,A -90.000,B 90.000,C 0.000} C_DIS
LIN {X -32.444,Y -19.308,Z -34.175,A -90.000,B 90.000,C 0.000} C_DIS
LIN {X -32.169,Y -19.308,Z -34.203,A -90.000,B 90.000,C 0.000} C_DIS
LIN {X -31.014,Y -19.308,Z -34.343,A -90.000,B 90.000,C 0.000} C_DIS
LIN {X -29.694,Y -19.308,Z -34.532,A -90.000,B 90.000,C 0.000} C_DIS
LIN {X -28.660,Y -19.308,Z -34.664,A -90.000,B 90.000,C 0.000} C_DIS
LIN {X -27.441,Y -19.308,Z -34.839,A -90.000,B 90.000,C 0.000} C_DIS
LIN {X -25.900,Y -19.308,Z -35.018,A -90.000,B 90.000,C 0.000} C_DIS
LIN {X -25.216,Y -19.308,Z -35.126,A -90.000,B 90.000,C 0.000} C_DIS
LIN {X -23.059,Y -19.308,Z -35.458,A -90.000,B 90.000,C 0.000} C_DIS
LIN {X -20.685,Y -19.308,Z -35.811,A -90.000,B 90.000,C 0.000} C_DIS
LIN {X -19.529,Y -19.308,Z -36.007,A -90.000,B 90.000,C 0.000} C_DIS
LIN {X -17.988,Y -19.308,Z -36.324,A -90.000,B 90.000,C 0.000} C_DIS
LIN {X -15.506,Y -19.308,Z -36.894,A -90.000,B 90.000,C 0.000} C_DIS
LIN {X -15.164,Y -19.308,Z -36.973,A -90.000,B 90.000,C 0.000} C_DIS
LIN {X -13.295,Y -19.308,Z -37.468,A -90.000,B 90.000,C 0.000} C_DIS
LIN {X -12.515,Y -19.308,Z -37.687,A -90.000,B 90.000,C 0.000} C_DIS
LIN {X -11.884,Y -19.308,Z -37.861,A -90.000,B 90.000,C 0.000} C_DIS
LIN {X -10.846,Y -19.308,Z -38.182,A -90.000,B 90.000,C 0.000} C_DIS
LIN {X -8.711,Y -19.308,Z -38.833,A -90.000,B 90.000,C 0.000} C_DIS
LIN {X -7.264,Y -19.308,Z -39.318,A -90.000,B 90.000,C 0.000} C_DIS
LIN {X -5.608,Y -19.308,Z -39.848,A -90.000,B 90.000,C 0.000} C_DIS
LIN {X -5.251,Y -19.308,Z -39.969,A -90.000,B 90.000,C 0.000} C_DIS
LIN {X -3.968,Y -19.308,Z -40.344,A -90.000,B 90.000,C 0.000} C_DIS
LIN {X -3.457,Y -19.308,Z -40.462,A -90.000,B 90.000,C 0.000} C_DIS
LIN {X -2.644,Y -19.308,Z -40.618,A -90.000,B 90.000,C 0.000} C_DIS
LIN {X -1.277,Y -19.308,Z -40.775,A -90.000,B 90.000,C 0.000} C_DIS
LIN {X 0.348,Y -19.308,Z -40.851,A -90.000,B 90.000,C 0.000} C_DIS
LIN {X 0.929,Y -19.308,Z -40.884,A -90.000,B 90.000,C 0.000} C_DIS
LIN {X 3.251,Y -19.308,Z -40.936,A -90.000,B 90.000,C 0.000} C_DIS
LIN {X 5.489,Y -19.308,Z -40.961,A -90.000,B 90.000,C 0.000} C_DIS
LIN {X 5.642,Y -19.308,Z -40.960,A -90.000,B 90.000,C 0.000} C_DIS
LIN {X 5.846,Y -19.308,Z -40.963,A -90.000,B 90.000,C 0.000} C_DIS
LIN {X 7.722,Y -19.308,Z -41.018,A -90.000,B 90.000,C 0.000} C_DIS
LIN {X 7.965,Y -19.308,Z -41.036,A -90.000,B 90.000,C 0.000} C_DIS
LIN {X 10.316,Y -19.308,Z -41.179,A -90.000,B 90.000,C 0.000} C_DIS
LIN {X 10.579,Y -19.308,Z -41.201,A -90.000,B 90.000,C 0.000} C_DIS
LIN {X 10.616,Y -19.308,Z -41.206,A -90.000,B 90.000,C 0.000} C_DIS
LIN {X 12.812,Y -19.308,Z -41.364,A -90.000,B 90.000,C 0.000} C_DIS
LIN {X 15.334,Y -19.308,Z -41.537,A -90.000,B 90.000,C 0.000} C_DIS
LIN {X 16.209,Y -19.308,Z -41.584,A -90.000,B 90.000,C 0.000} C_DIS
LIN {X 17.519,Y -19.308,Z -41.641,A -90.000,B 90.000,C 0.000} C_DIS
LIN {X 19.899,Y -19.308,Z -41.670,A -90.000,B 90.000,C 0.000} C_DIS
LIN {X 20.003,Y -19.308,Z -41.670,A -90.000,B 90.000,C 0.000} C_DIS
LIN {X 22.157,Y -19.308,Z -41.570,A -90.000,B 90.000,C 0.000} C_DIS
LIN {X 23.011,Y -19.308,Z -41.484,A -90.000,B 90.000,C 0.000} C_DIS
LIN {X 24.203,Y -19.308,Z -41.332,A -90.000,B 90.000,C 0.000} C_DIS
LIN {X 25.024,Y -19.308,Z -41.179,A -90.000,B 90.000,C 0.000} C_DIS
LIN {X 26.034,Y -19.308,Z -41.003,A -90.000,B 90.000,C 0.000} C_DIS
LIN {X 26.385,Y -19.308,Z -40.918,A -90.000,B 90.000,C 0.000} C_DIS
LIN {X 27.005,Y -19.308,Z -40.781,A -90.000,B 90.000,C 0.000} C_DIS
LIN {X 27.684,Y -19.308,Z -40.627,A -90.000,B 90.000,C 0.000} C_DIS
LIN {X 28.084,Y -19.308,Z -40.555,A -90.000,B 90.000,C 0.000} C_DIS
LIN {X 29.000,Y -19.308,Z -40.316,A -90.000,B 90.000,C 0.000} C_DIS
LIN {X 30.180,Y -19.308,Z -40.073,A -90.000,B 90.000,C 0.000} C_DIS
LIN {X 30.447,Y -19.308,Z -39.998,A -90.000,B 90.000,C 0.000} C_DIS
LIN {X 31.331,Y -19.308,Z -39.805,A -90.000,B 90.000,C 0.000} C_DIS
LIN {X 31.829,Y -19.308,Z -39.699,A -90.000,B 90.000,C 0.000} C_DIS
LIN {X 32.248,Y -19.308,Z -39.620,A -90.000,B 90.000,C 0.000} C_DIS
LIN {X 32.694,Y -19.308,Z -39.558,A -90.000,B 90.000,C 0.000} C_DIS
LIN {X 33.805,Y -19.308,Z -39.322,A -90.000,B 90.000,C 0.000} C_DIS
LIN {X 35.232,Y -19.308,Z -39.127,A -90.000,B 90.000,C 0.000} C_DIS
LIN {X 35.274,Y -19.308,Z -39.120,A -90.000,B 90.000,C 0.000} C_DIS
LIN {X 35.843,Y -19.308,Z -39.045,A -90.000,B 90.000,C 0.000} C_DIS
LIN {X 36.645,Y -19.308,Z -38.970,A -90.000,B 90.000,C 0.000} C_DIS
LIN {X 36.922,Y -19.308,Z -38.946,A -90.000,B 90.000,C 0.000} C_DIS
LIN {X 37.835,Y -19.308,Z -38.875,A -90.000,B 90.000,C 0.000} C_DIS
LIN {X 38.404,Y -19.308,Z -38.868,A -90.000,B 90.000,C 0.000} C_DIS
LIN {X 38.678,Y -19.308,Z -38.871,A -90.000,B 90.000,C 0.000} C_DIS
LIN {X 39.964,Y -19.308,Z -38.871,A -90.000,B 90.000,C 0.000} C_DIS
LIN {X 40.439,Y -19.308,Z -38.895,A -90.000,B 90.000,C 0.000} C_DIS
LIN {X 42.166,Y -19.308,Z -39.043,A -90.000,B 90.000,C 0.000} C_DIS
LIN {X 42.598,Y -19.308,Z -39.097,A -90.000,B 90.000,C 0.000} C_DIS
LIN {X 43.073,Y -19.308,Z -39.180,A -90.000,B 90.000,C 0.000} C_DIS
LIN {X 43.615,Y -19.308,Z -39.280,A -90.000,B 90.000,C 0.000} C_DIS
LIN {X 44.751,Y -19.308,Z -39.521,A -90.000,B 90.000,C 0.000} C_DIS
LIN {X 45.611,Y -19.308,Z -39.729,A -90.000,B 90.000,C 0.000} C_DIS
LIN {X 46.078,Y -19.308,Z -39.867,A -90.000,B 90.000,C 0.000} C_DIS
LIN {X 47.370,Y -19.308,Z -40.318,A -90.000,B 90.000,C 0.000} C_DIS
LIN {X 49.021,Y -19.308,Z -40.962,A -90.000,B 90.000,C 0.000} C_DIS
LIN {X 49.434,Y -19.308,Z -41.131,A -90.000,B 90.000,C 0.000} C_DIS
LIN {X 49.569,Y -19.308,Z -41.195,A -90.000,B 90.000,C 0.000} C_DIS
LIN {X 50.058,Y -19.308,Z -41.439,A -90.000,B 90.000,C 0.000} C_DIS
LIN {X 50.943,Y -19.308,Z -41.885,A -90.000,B 90.000,C 0.000} C_DIS
LIN {X 52.074,Y -19.308,Z -42.483,A -90.000,B 90.000,C 0.000} C_DIS
LIN {X 52.542,Y -19.308,Z -42.736,A -90.000,B 90.000,C 0.000} C_DIS
LIN {X 53.771,Y -19.308,Z -43.517,A -90.000,B 90.000,C 0.000} C_DIS
LIN {X 55.062,Y -19.308,Z -44.321,A -90.000,B 90.000,C 0.000} C_DIS
LIN {X 55.465,Y -19.308,Z -44.596,A -90.000,B 90.000,C 0.000} C_DIS
LIN {X 55.826,Y -19.308,Z -44.867,A -90.000,B 90.000,C 0.000} C_DIS
LIN {X 56.618,Y -19.308,Z -45.438,A -90.000,B 90.000,C 0.000} C_DIS
LIN {X 57.734,Y -19.308,Z -46.268,A -90.000,B 90.000,C 0.000} C_DIS
LIN {X 58.903,Y -19.308,Z -47.255,A -90.000,B 90.000,C 0.000} C_DIS
LIN {X 60.100,Y -19.308,Z -48.291,A -90.000,B 90.000,C 0.000} C_DIS
LIN {X 61.796,Y -19.308,Z -49.795,A -90.000,B 90.000,C 0.000} C_DIS
LIN {X 62.592,Y -19.308,Z -50.440,A -90.000,B 90.000,C 0.000} C_DIS
LIN {X 62.965,Y -19.308,Z -50.753,A -90.000,B 90.000,C 0.000} C_DIS
LIN {X 63.487,Y -19.308,Z -51.195,A -90.000,B 90.000,C 0.000} C_DIS
LIN {X 64.755,Y -19.308,Z -52.118,A -90.000,B 90.000,C 0.000} C_DIS
LIN {X 65.190,Y -19.308,Z -52.427,A -90.000,B 90.000,C 0.000} C_DIS
LIN {X 66.037,Y -19.308,Z -52.952,A -90.000,B 90.000,C 0.000} C_DIS
LIN {X 67.690,Y -19.308,Z -53.920,A -90.000,B 90.000,C 0.000} C_DIS
LIN {X 69.402,Y -19.308,Z -54.896,A -90.000,B 90.000,C 0.000} C_DIS
LIN {X 71.579,Y -19.308,Z -56.188,A -90.000,B 90.000,C 0.000} C_DIS
LIN {X 73.583,Y -19.308,Z -57.508,A -90.000,B 90.000,C 0.000} C_DIS
LIN {X 73.985,Y -19.308,Z -57.775,A -90.000,B 90.000,C 0.000} C_DIS
LIN {X 75.186,Y -19.308,Z -58.727,A -90.000,B 90.000,C 0.000} C_DIS
LIN {X 75.708,Y -19.308,Z -59.133,A -90.000,B 90.000,C 0.000} C_DIS
LIN {X 76.080,Y -19.308,Z -59.440,A -90.000,B 90.000,C 0.000} C_DIS
LIN {X 76.981,Y -19.308,Z -60.280,A -90.000,B 90.000,C 0.000} C_DIS
LIN {X 77.535,Y -19.308,Z -60.781,A -90.000,B 90.000,C 0.000} C_DIS
LIN {X 77.872,Y -19.308,Z -61.117,A -90.000,B 90.000,C 0.000} C_DIS
LIN {X 78.140,Y -19.308,Z -61.405,A -90.000,B 90.000,C 0.000} C_DIS
LIN {X 78.585,Y -19.308,Z -61.865,A -90.000,B 90.000,C 0.000} C_DIS
LIN {X 78.930,Y -19.308,Z -62.217,A -90.000,B 90.000,C 0.000} C_DIS
LIN {X 79.232,Y -19.316,Z -62.529,A -90.000,B 90.000,C 0.000} C_DIS
LIN {X 79.359,Y -19.473,Z -62.677,A -90.000,B 90.000,C 0.000} C_DIS
LIN {X 79.361,Y -25.896,Z -62.679,A -90.000,B 90.000,C 0.000} C_DIS
LIN {X 79.368,Y -26.127,Z -62.685,A -90.000,B 90.000,C 0.000} C_DIS
LIN {X 79.376,Y -26.270,Z -62.694,A -90.000,B 90.000,C 0.000} C_DIS
LIN {X 79.392,Y -26.461,Z -62.710,A -90.000,B 90.000,C 0.000} C_DIS
LIN {X 79.425,Y -26.767,Z -62.742,A -90.000,B 90.000,C 0.000} C_DIS
LIN {X 79.488,Y -27.181,Z -62.805,A -90.000,B 90.000,C 0.000} C_DIS
LIN {X 79.607,Y -27.691,Z -62.923,A -90.000,B 90.000,C 0.000} C_DIS
LIN {X 79.717,Y -28.042,Z -63.030,A -90.000,B 90.000,C 0.000} C_DIS
LIN {X 79.820,Y -28.312,Z -63.127,A -90.000,B 90.000,C 0.000} C_DIS
LIN {X 79.914,Y -28.543,Z -63.214,A -90.000,B 90.000,C 0.000} C_DIS
LIN {X 80.081,Y -28.906,Z -63.358,A -90.000,B 90.000,C 0.000} C_DIS
LIN {X 80.153,Y -29.050,Z -63.415,A -90.000,B 90.000,C 0.000} C_DIS
LIN {X 80.219,Y -29.170,Z -63.463,A -90.000,B 90.000,C 0.000} C_DIS
LIN {X 80.305,Y -29.314,Z -63.518,A -90.000,B 90.000,C 0.000} C_DIS
LIN {X 80.354,Y -29.388,Z -63.542,A -90.000,B 90.000,C 0.000} C_DIS
LIN {X 80.397,Y -29.447,Z -63.558,A -90.000,B 90.000,C 0.000} C_DIS
LIN {X 80.416,Y -29.472,Z -63.562,A -90.000,B 90.000,C 0.000} C_DIS
LIN {X 80.451,Y -29.514,Z -63.564,A -90.000,B 90.000,C 0.000} C_DIS
LIN {X 80.480,Y -29.545,Z -63.557,A -90.000,B 90.000,C 0.000} C_DIS
LIN {X 80.505,Y -29.567,Z -63.542,A -90.000,B 90.000,C 0.000} C_DIS
LIN {X 80.526,Y -29.580,Z -63.518,A -90.000,B 90.000,C 0.000} C_DIS
LIN {X 80.534,Y -29.583,Z -63.503,A -90.000,B 90.000,C 0.000} C_DIS
LIN {X 80.549,Y -29.584,Z -63.467,A -90.000,B 90.000,C 0.000} C_DIS
LIN {X 80.560,Y -29.577,Z -63.424,A -90.000,B 90.000,C 0.000} C_DIS
LIN {X 80.570,Y -29.554,Z -63.343,A -90.000,B 90.000,C 0.000} C_DIS
LIN {X 80.573,Y -29.530,Z -63.280,A -90.000,B 90.000,C 0.000} C_DIS
LIN {X 80.571,Y -29.464,Z -63.132,A -90.000,B 90.000,C 0.000} C_DIS
LIN {X 80.567,Y -29.422,Z -63.047,A -90.000,B 90.000,C 0.000} C_DIS
LIN {X 80.554,Y -29.319,Z -62.856,A -90.000,B 90.000,C 0.000} C_DIS
LIN {X 80.517,Y -29.047,Z -62.398,A -90.000,B 90.000,C 0.000} C_DIS
LIN {X 80.497,Y -28.872,Z -62.132,A -90.000,B 90.000,C 0.000} C_DIS
LIN {X 80.480,Y -28.674,Z -61.842,A -90.000,B 90.000,C 0.000} C_DIS
LIN {X 80.468,Y -28.454,Z -61.531,A -90.000,B 90.000,C 0.000} C_DIS
LIN {X 80.462,Y -28.223,Z -61.199,A -90.000,B 90.000,C 0.000} C_DIS
LIN {X 80.466,Y -27.987,Z -60.847,A -90.000,B 90.000,C 0.000} C_DIS
LIN {X 80.473,Y -27.858,Z -60.664,A -90.000,B 90.000,C 0.000} C_DIS
LIN {X 80.482,Y -27.720,Z -60.476,A -90.000,B 90.000,C 0.000} C_DIS
LIN {X 80.496,Y -27.570,Z -60.285,A -90.000,B 90.000,C 0.000} C_DIS
LIN {X 80.513,Y -27.407,Z -60.089,A -90.000,B 90.000,C 0.000} C_DIS
LIN {X 80.546,Y -27.133,Z -59.787,A -90.000,B 90.000,C 0.000} C_DIS
LIN {X 80.560,Y -27.045,Z -59.685,A -90.000,B 90.000,C 0.000} C_DIS
LIN {X 80.590,Y -26.873,Z -59.477,A -90.000,B 90.000,C 0.000} C_DIS
LIN {X 80.646,Y -26.659,Z -59.159,A -90.000,B 90.000,C 0.000} C_DIS
LIN {X 80.690,Y -26.510,Z -58.942,A -90.000,B 90.000,C 0.000} C_DIS
LIN {X 80.739,Y -26.352,Z -58.723,A -90.000,B 90.000,C 0.000} C_DIS
LIN {X 80.795,Y -26.183,Z -58.500,A -90.000,B 90.000,C 0.000} C_DIS
LIN {X 80.825,Y -26.091,Z -58.388,A -90.000,B 90.000,C 0.000} C_DIS
LIN {X 80.857,Y -25.990,Z -58.275,A -90.000,B 90.000,C 0.000} C_DIS
LIN {X 80.891,Y -25.869,Z -58.161,A -90.000,B 90.000,C 0.000} C_DIS
LIN {X 80.908,Y -25.785,Z -58.104,A -90.000,B 90.000,C 0.000} C_DIS
LIN {X 80.917,Y -25.720,Z -58.075,A -90.000,B 90.000,C 0.000} C_DIS
LIN {X 80.919,Y -25.693,Z -58.068,A -90.000,B 90.000,C 0.000} C_DIS
LIN {X 80.921,Y -25.647,Z -58.062,A -90.000,B 90.000,C 0.000} C_DIS
LIN {X 80.921,Y -19.666,Z -58.061,A -90.000,B 90.000,C 0.000} C_DIS
LIN {X 80.963,Y -19.574,Z -57.931,A -90.000,B 90.000,C 0.000} C_DIS
LIN {X 81.002,Y -19.446,Z -57.815,A -90.000,B 90.000,C 0.000} C_DIS
LIN {X 81.022,Y -19.334,Z -57.757,A -90.000,B 90.000,C 0.000} C_DIS
LIN {X 81.042,Y -19.308,Z -57.699,A -90.000,B 90.000,C 0.000} C_DIS
LIN {X 81.094,Y -19.307,Z -57.585,A -90.000,B 90.000,C 0.000} C_DIS
LIN {X 81.231,Y -19.307,Z -57.230,A -90.000,B 90.000,C 0.000} C_DIS
LIN {X 81.281,Y -19.308,Z -57.111,A -90.000,B 90.000,C 0.000} C_DIS
LIN {X 81.339,Y -19.308,Z -56.994,A -90.000,B 90.000,C 0.000} C_DIS
LIN {X 81.700,Y -19.308,Z -56.182,A -90.000,B 90.000,C 0.000} C_DIS
LIN {X 82.142,Y -19.308,Z -55.092,A -90.000,B 90.000,C 0.000} C_DIS
LIN {X 82.335,Y -19.308,Z -54.666,A -90.000,B 90.000,C 0.000} C_DIS
LIN {X 83.331,Y -19.308,Z -52.811,A -90.000,B 90.000,C 0.000} C_DIS
LIN {X 83.577,Y -19.308,Z -52.389,A -90.000,B 90.000,C 0.000} C_DIS
LIN {X 84.750,Y -19.308,Z -50.667,A -90.000,B 90.000,C 0.000} C_DIS
LIN {X 85.025,Y -19.308,Z -50.291,A -90.000,B 90.000,C 0.000} C_DIS
LIN {X 86.337,Y -19.308,Z -48.714,A -90.000,B 90.000,C 0.000} C_DIS
LIN {X 86.664,Y -19.308,Z -48.352,A -90.000,B 90.000,C 0.000} C_DIS
LIN {X 88.117,Y -19.308,Z -46.880,A -90.000,B 90.000,C 0.000} C_DIS
LIN {X 88.479,Y -19.308,Z -46.553,A -90.000,B 90.000,C 0.000} C_DIS
LIN {X 90.061,Y -19.308,Z -45.164,A -90.000,B 90.000,C 0.000} C_DIS
LIN {X 91.740,Y -19.308,Z -43.859,A -90.000,B 90.000,C 0.000} C_DIS
LIN {X 92.110,Y -19.308,Z -43.588,A -90.000,B 90.000,C 0.000} C_DIS
LIN {X 93.780,Y -19.308,Z -42.419,A -90.000,B 90.000,C 0.000} C_DIS
LIN {X 95.447,Y -19.308,Z -41.365,A -90.000,B 90.000,C 0.000} C_DIS
LIN {X 95.948,Y -19.308,Z -41.073,A -90.000,B 90.000,C 0.000} C_DIS
LIN {X 97.376,Y -19.308,Z -40.260,A -90.000,B 90.000,C 0.000} C_DIS
LIN {X 98.805,Y -19.308,Z -39.523,A -90.000,B 90.000,C 0.000} C_DIS
LIN {X 100.266,Y -19.308,Z -38.830,A -90.000,B 90.000,C 0.000} C_DIS
LIN {X 102.148,Y -19.308,Z -37.978,A -90.000,B 90.000,C 0.000} C_DIS
LIN {X 103.348,Y -19.308,Z -37.442,A -90.000,B 90.000,C 0.000} C_DIS
LIN {X 103.753,Y -19.308,Z -37.262,A -90.000,B 90.000,C 0.000} C_DIS
LIN {X 104.475,Y -19.308,Z -36.943,A -90.000,B 90.000,C 0.000} C_DIS
LIN {X 105.369,Y -19.308,Z -36.566,A -90.000,B 90.000,C 0.000} C_DIS
LIN {X 106.900,Y -19.308,Z -35.958,A -90.000,B 90.000,C 0.000} C_DIS
LIN {X 107.422,Y -19.308,Z -35.760,A -90.000,B 90.000,C 0.000} C_DIS
LIN {X 107.855,Y -19.308,Z -35.604,A -90.000,B 90.000,C 0.000} C_DIS
LIN {X 108.317,Y -19.308,Z -35.448,A -90.000,B 90.000,C 0.000} C_DIS
LIN {X 108.745,Y -19.308,Z -35.333,A -90.000,B 90.000,C 0.000} C_DIS
LIN {X 109.221,Y -19.308,Z -35.225,A -90.000,B 90.000,C 0.000} C_DIS
LIN {X 109.676,Y -19.308,Z -35.166,A -90.000,B 90.000,C 0.000} C_DIS
LIN {X 110.108,Y -19.308,Z -35.113,A -90.000,B 90.000,C 0.000} C_DIS
LIN {X 110.596,Y -19.308,Z -35.105,A -90.000,B 90.000,C 0.000} C_DIS
LIN {X 110.949,Y -19.308,Z -35.117,A -90.000,B 90.000,C 0.000} C_DIS
LIN {X 111.435,Y -19.308,Z -35.158,A -90.000,B 90.000,C 0.000} C_DIS
LIN {X 112.068,Y -19.308,Z -35.277,A -90.000,B 90.000,C 0.000} C_DIS
LIN {X 112.405,Y -19.308,Z -35.362,A -90.000,B 90.000,C 0.000} C_DIS
LIN {X 112.893,Y -19.308,Z -35.508,A -90.000,B 90.000,C 0.000} C_DIS
LIN {X 113.055,Y -19.308,Z -35.560,A -90.000,B 90.000,C 0.000} C_DIS
LIN {X 113.505,Y -19.308,Z -35.746,A -90.000,B 90.000,C 0.000} C_DIS
LIN {X 113.979,Y -19.308,Z -35.973,A -90.000,B 90.000,C 0.000} C_DIS
LIN {X 114.424,Y -19.308,Z -36.214,A -90.000,B 90.000,C 0.000} C_DIS
LIN {X 114.540,Y -19.308,Z -36.286,A -90.000,B 90.000,C 0.000} C_DIS
LIN {X 114.956,Y -19.308,Z -36.570,A -90.000,B 90.000,C 0.000} C_DIS
LIN {X 115.050,Y -19.308,Z -36.644,A -90.000,B 90.000,C 0.000} C_DIS
LIN {X 115.433,Y -19.308,Z -36.967,A -90.000,B 90.000,C 0.000} C_DIS
LIN {X 115.513,Y -19.308,Z -37.039,A -90.000,B 90.000,C 0.000} C_DIS
LIN {X 115.878,Y -19.308,Z -37.417,A -90.000,B 90.000,C 0.000} C_DIS
LIN {X 116.083,Y -19.308,Z -37.635,A -90.000,B 90.000,C 0.000} C_DIS
LIN {X 116.439,Y -19.308,Z -38.088,A -90.000,B 90.000,C 0.000} C_DIS
LIN {X 116.700,Y -19.308,Z -38.500,A -90.000,B 90.000,C 0.000} C_DIS
LIN {X 116.933,Y -19.308,Z -38.973,A -90.000,B 90.000,C 0.000} C_DIS
LIN {X 116.983,Y -19.308,Z -39.082,A -90.000,B 90.000,C 0.000} C_DIS
LIN {X 117.060,Y -19.308,Z -39.253,A -90.000,B 90.000,C 0.000} C_DIS
LIN {X 117.109,Y -19.308,Z -39.379,A -90.000,B 90.000,C 0.000} C_DIS
LIN {X 117.260,Y -19.308,Z -39.781,A -90.000,B 90.000,C 0.000} C_DIS
LIN {X 117.393,Y -19.308,Z -40.294,A -90.000,B 90.000,C 0.000} C_DIS
LIN {X 117.462,Y -19.308,Z -40.593,A -90.000,B 90.000,C 0.000} C_DIS
LIN {X 117.543,Y -19.308,Z -41.125,A -90.000,B 90.000,C 0.000} C_DIS
LIN {X 117.593,Y -19.308,Z -41.494,A -90.000,B 90.000,C 0.000} C_DIS
LIN {X 117.630,Y -19.308,Z -41.874,A -90.000,B 90.000,C 0.000} C_DIS
LIN {X 117.657,Y -19.308,Z -42.399,A -90.000,B 90.000,C 0.000} C_DIS
LIN {X 117.668,Y -19.308,Z -42.703,A -90.000,B 90.000,C 0.000} C_DIS
LIN {X 117.664,Y -19.308,Z -42.881,A -90.000,B 90.000,C 0.000} C_DIS
LIN {X 117.651,Y -19.308,Z -43.202,A -90.000,B 90.000,C 0.000} C_DIS
LIN {X 117.606,Y -19.308,Z -43.738,A -90.000,B 90.000,C 0.000} C_DIS
LIN {X 117.567,Y -19.308,Z -44.117,A -90.000,B 90.000,C 0.000} C_DIS
LIN {X 117.489,Y -19.308,Z -44.635,A -90.000,B 90.000,C 0.000} C_DIS
LIN {X 117.399,Y -19.308,Z -45.114,A -90.000,B 90.000,C 0.000} C_DIS
LIN {X 117.260,Y -19.308,Z -45.739,A -90.000,B 90.000,C 0.000} C_DIS
LIN {X 117.095,Y -19.308,Z -46.292,A -90.000,B 90.000,C 0.000} C_DIS
LIN {X 116.900,Y -19.308,Z -46.938,A -90.000,B 90.000,C 0.000} C_DIS
LIN {X 116.538,Y -19.308,Z -47.876,A -90.000,B 90.000,C 0.000} C_DIS
LIN {X 116.372,Y -19.308,Z -48.278,A -90.000,B 90.000,C 0.000} C_DIS
LIN {X 115.873,Y -19.308,Z -49.350,A -90.000,B 90.000,C 0.000} C_DIS
LIN {X 115.208,Y -19.308,Z -50.679,A -90.000,B 90.000,C 0.000} C_DIS
LIN {X 114.622,Y -19.308,Z -51.838,A -90.000,B 90.000,C 0.000} C_DIS
LIN {X 113.941,Y -19.308,Z -53.229,A -90.000,B 90.000,C 0.000} C_DIS
LIN {X 113.276,Y -19.308,Z -54.687,A -90.000,B 90.000,C 0.000} C_DIS
LIN {X 112.799,Y -19.308,Z -55.830,A -90.000,B 90.000,C 0.000} C_DIS
LIN {X 112.213,Y -19.308,Z -57.388,A -90.000,B 90.000,C 0.000} C_DIS
LIN {X 111.674,Y -19.308,Z -59.009,A -90.000,B 90.000,C 0.000} C_DIS
LIN {X 111.260,Y -19.308,Z -60.445,A -90.000,B 90.000,C 0.000} C_DIS
LIN {X 110.736,Y -19.308,Z -62.369,A -90.000,B 90.000,C 0.000} C_DIS
LIN {X 110.147,Y -19.308,Z -64.456,A -90.000,B 90.000,C 0.000} C_DIS
LIN {X 110.102,Y -19.308,Z -64.608,A -90.000,B 90.000,C 0.000} C_DIS
LIN {X 110.021,Y -19.308,Z -64.879,A -90.000,B 90.000,C 0.000} C_DIS
LIN {X 109.345,Y -19.308,Z -67.050,A -90.000,B 90.000,C 0.000} C_DIS
LIN {X 108.519,Y -19.308,Z -69.358,A -90.000,B 90.000,C 0.000} C_DIS
LIN {X 107.573,Y -19.308,Z -71.738,A -90.000,B 90.000,C 0.000} C_DIS
LIN {X 107.403,Y -19.308,Z -72.150,A -90.000,B 90.000,C 0.000} C_DIS
LIN {X 106.414,Y -19.308,Z -74.420,A -90.000,B 90.000,C 0.000} C_DIS
LIN {X 105.411,Y -19.308,Z -76.516,A -90.000,B 90.000,C 0.000} C_DIS
LIN {X 104.209,Y -19.308,Z -78.763,A -90.000,B 90.000,C 0.000} C_DIS
